//     Term 143 (AT2000-0250)/Term 144 (AT2000-5250)/FB Inputs/Value Channel 06 <-> Data Pointer/RawPositionValues[5]
//     Term 143 (AT2000-0250)/Term 144 (AT2000-5250)/FB Inputs/Value Channel 07 <-> Data Pointer/RawPositionValues[6]
//     Term 143 (AT2000-0250)/Term 144 (AT2000-5250)/FB Inputs/Value Channel 08 <-> Data Pointer/RawPositionValues[7]
//     Term 143 (AT2000-0250)/Term 144 (AT2000-5250)/FB Inputs/Value Channel 09 <-> Data Pointer/RawPositionValues[8]
//     Term 143 (AT2000-0250)/Term 144 (AT2000-5250)/FB Inputs/Value Channel 10 <-> Data Pointer/RawPositionValues[9]
//     Term 143 (AT2000-0250)/Term 144 (AT2000-5250)/FB Inputs/Value Channel 11 <-> Data Pointer/RawPositionValues[10]
//     Term 143 (AT2000-0250)/Term 144 (AT2000-5250)/FB Inputs/Value Channel 12 <-> Data Pointer/RawPositionValues[11]
//     Term 143 (AT2000-0250)/Term 144 (AT2000-5250)/FB Inputs/Value Channel 13 <-> Data Pointer/RawPositionValues[12]
//     Term 143 (AT2000-0250)/Term 144 (AT2000-5250)/FB Inputs/Value Channel 14 <-> Data Pointer/RawPositionValues[13]
//     Term 143 (AT2000-0250)/Term 144 (AT2000-5250)/FB Inputs/Value Channel 15 <-> Data Pointer/RawPositionValues[14]
//     Term 143 (AT2000-0250)/Term 144 (AT2000-5250)/FB Inputs/Value Channel 16 <-> Data Pointer/RawPositionValues[15]
//     Term 143 (AT2000-0250)/Term 144 (AT2000-5250)/FB Inputs/Value Channel 17 <-> Data Pointer/RawPositionValues[16]
//     Term 143 (AT2000-0250)/Term 144 (AT2000-5250)/FB Inputs/Value Channel 18 <-> Data Pointer/RawPositionValues[17]
//     Term 143 (AT2000-0250)/Term 144 (AT2000-5250)/FB Inputs/Value Channel 19 <-> Data Pointer/RawPositionValues[18]
//     Term 143 (AT2000-0250)/Term 144 (AT2000-5250)/FB Inputs/Value Channel 20 <-> Data Pointer/RawPositionValues[19]
//     Term 143 (AT2000-0250)/Term 144 (AT2000-5250)/FB Inputs/Value Channel 21 <-> Data Pointer/RawPositionValues[20]
//     Term 143 (AT2000-0250)/Term 144 (AT2000-5250)/FB Inputs/Value Channel 22 <-> Data Pointer/RawPositionValues[21]
//     Term 143 (AT2000-0250)/Term 144 (AT2000-5250)/FB Inputs/Value Channel 23 <-> Data Pointer/RawPositionValues[22]
//     Term 143 (AT2000-0250)/Term 144 (AT2000-5250)/FB Inputs/Value Channel 24 <-> Data Pointer/RawPositionValues[23]
//     Term 143 (AT2000-0250)/Term 144 (AT2000-5250)/FB Inputs/Value Channel 25 <-> Data Pointer/RawPositionValues[24]
//     Term 143 (AT2000-0250)/Term 144 (AT2000-5250)/FB Inputs/Value Channel 26 <-> Data Pointer/RawPositionValues[25]
//     Term 143 (AT2000-0250)/Term 144 (AT2000-5250)/FB Inputs/Value Channel 27 <-> Data Pointer/RawPositionValues[26]
//     Term 143 (AT2000-0250)/Term 144 (AT2000-5250)/FB Inputs/Value Channel 28 <-> Data Pointer/RawPositionValues[27]
//     Term 143 (AT2000-0250)/Term 144 (AT2000-5250)/FB Inputs/Value Channel 29 <-> Data Pointer/RawPositionValues[28]
//     Term 143 (AT2000-0250)/Term 144 (AT2000-5250)/FB Inputs/Value Channel 30 <-> Data Pointer/RawPositionValues[29]
//     Term 143 (AT2000-0250)/Term 144 (AT2000-5250)/FB Inputs/Value Channel 31 <-> Data Pointer/RawPositionValues[30]
//     Term 143 (AT2000-0250)/Term 144 (AT2000-5250)/FB Inputs/Value Channel 32 <-> Data Pointer/RawPositionValues[31]
//   Device 17 <-> TcCOM Objects/XTS ProcessingUnit 1/Part 1/Module 73
//     Term 145 (AT2000-0250)/CC Inputs/Current actual value Ch.1 <-> Data Pointer/CurrentActualValues[0]
//     Term 145 (AT2000-0250)/CC Inputs/Current actual value Ch.10 <-> Data Pointer/CurrentActualValues[9]
//     Term 145 (AT2000-0250)/CC Inputs/Current actual value Ch.11 <-> Data Pointer/CurrentActualValues[10]
//     Term 145 (AT2000-0250)/CC Inputs/Current actual value Ch.12 <-> Data Pointer/CurrentActualValues[11]
//     Term 145 (AT2000-0250)/CC Inputs/Current actual value Ch.13 <-> Data Pointer/CurrentActualValues[12]
//     Term 145 (AT2000-0250)/CC Inputs/Current actual value Ch.14 <-> Data Pointer/CurrentActualValues[13]
//     Term 145 (AT2000-0250)/CC Inputs/Current actual value Ch.15 <-> Data Pointer/CurrentActualValues[14]
//     Term 145 (AT2000-0250)/CC Inputs/Current actual value Ch.2 <-> Data Pointer/CurrentActualValues[1]
//     Term 145 (AT2000-0250)/CC Inputs/Current actual value Ch.3 <-> Data Pointer/CurrentActualValues[2]
//     Term 145 (AT2000-0250)/CC Inputs/Current actual value Ch.4 <-> Data Pointer/CurrentActualValues[3]
//     Term 145 (AT2000-0250)/CC Inputs/Current actual value Ch.5 <-> Data Pointer/CurrentActualValues[4]
//     Term 145 (AT2000-0250)/CC Inputs/Current actual value Ch.6 <-> Data Pointer/CurrentActualValues[5]
//     Term 145 (AT2000-0250)/CC Inputs/Current actual value Ch.7 <-> Data Pointer/CurrentActualValues[6]
//     Term 145 (AT2000-0250)/CC Inputs/Current actual value Ch.8 <-> Data Pointer/CurrentActualValues[7]
//     Term 145 (AT2000-0250)/CC Inputs/Current actual value Ch.9 <-> Data Pointer/CurrentActualValues[8]
//     Term 145 (AT2000-0250)/CC Inputs/Status <-> Data Pointer/Status
//     Term 145 (AT2000-0250)/CC Outputs/Control <-> Data Pointer/Control
//     Term 145 (AT2000-0250)/CC Outputs/Current setpoint value Ch.1 <-> Data Pointer/CurrentSetpointValues[0]
//     Term 145 (AT2000-0250)/CC Outputs/Current setpoint value Ch.10 <-> Data Pointer/CurrentSetpointValues[9]
//     Term 145 (AT2000-0250)/CC Outputs/Current setpoint value Ch.11 <-> Data Pointer/CurrentSetpointValues[10]
//     Term 145 (AT2000-0250)/CC Outputs/Current setpoint value Ch.12 <-> Data Pointer/CurrentSetpointValues[11]
//     Term 145 (AT2000-0250)/CC Outputs/Current setpoint value Ch.13 <-> Data Pointer/CurrentSetpointValues[12]
//     Term 145 (AT2000-0250)/CC Outputs/Current setpoint value Ch.14 <-> Data Pointer/CurrentSetpointValues[13]
//     Term 145 (AT2000-0250)/CC Outputs/Current setpoint value Ch.15 <-> Data Pointer/CurrentSetpointValues[14]
//     Term 145 (AT2000-0250)/CC Outputs/Current setpoint value Ch.2 <-> Data Pointer/CurrentSetpointValues[1]
//     Term 145 (AT2000-0250)/CC Outputs/Current setpoint value Ch.3 <-> Data Pointer/CurrentSetpointValues[2]
//     Term 145 (AT2000-0250)/CC Outputs/Current setpoint value Ch.4 <-> Data Pointer/CurrentSetpointValues[3]
//     Term 145 (AT2000-0250)/CC Outputs/Current setpoint value Ch.5 <-> Data Pointer/CurrentSetpointValues[4]
//     Term 145 (AT2000-0250)/CC Outputs/Current setpoint value Ch.6 <-> Data Pointer/CurrentSetpointValues[5]
//     Term 145 (AT2000-0250)/CC Outputs/Current setpoint value Ch.7 <-> Data Pointer/CurrentSetpointValues[6]
//     Term 145 (AT2000-0250)/CC Outputs/Current setpoint value Ch.8 <-> Data Pointer/CurrentSetpointValues[7]
//     Term 145 (AT2000-0250)/CC Outputs/Current setpoint value Ch.9 <-> Data Pointer/CurrentSetpointValues[8]
//     Term 145 (AT2000-0250)/Term 146 (AT2000-5250)/FB Inputs/Value Channel 01 <-> Data Pointer/RawPositionValues[0]
//     Term 145 (AT2000-0250)/Term 146 (AT2000-5250)/FB Inputs/Value Channel 02 <-> Data Pointer/RawPositionValues[1]
//     Term 145 (AT2000-0250)/Term 146 (AT2000-5250)/FB Inputs/Value Channel 03 <-> Data Pointer/RawPositionValues[2]
//     Term 145 (AT2000-0250)/Term 146 (AT2000-5250)/FB Inputs/Value Channel 04 <-> Data Pointer/RawPositionValues[3]
//     Term 145 (AT2000-0250)/Term 146 (AT2000-5250)/FB Inputs/Value Channel 05 <-> Data Pointer/RawPositionValues[4]
//     Term 145 (AT2000-0250)/Term 146 (AT2000-5250)/FB Inputs/Value Channel 06 <-> Data Pointer/RawPositionValues[5]
//     Term 145 (AT2000-0250)/Term 146 (AT2000-5250)/FB Inputs/Value Channel 07 <-> Data Pointer/RawPositionValues[6]
//     Term 145 (AT2000-0250)/Term 146 (AT2000-5250)/FB Inputs/Value Channel 08 <-> Data Pointer/RawPositionValues[7]
//     Term 145 (AT2000-0250)/Term 146 (AT2000-5250)/FB Inputs/Value Channel 09 <-> Data Pointer/RawPositionValues[8]
//     Term 145 (AT2000-0250)/Term 146 (AT2000-5250)/FB Inputs/Value Channel 10 <-> Data Pointer/RawPositionValues[9]
//     Term 145 (AT2000-0250)/Term 146 (AT2000-5250)/FB Inputs/Value Channel 11 <-> Data Pointer/RawPositionValues[10]
//     Term 145 (AT2000-0250)/Term 146 (AT2000-5250)/FB Inputs/Value Channel 12 <-> Data Pointer/RawPositionValues[11]
//     Term 145 (AT2000-0250)/Term 146 (AT2000-5250)/FB Inputs/Value Channel 13 <-> Data Pointer/RawPositionValues[12]
//     Term 145 (AT2000-0250)/Term 146 (AT2000-5250)/FB Inputs/Value Channel 14 <-> Data Pointer/RawPositionValues[13]
//     Term 145 (AT2000-0250)/Term 146 (AT2000-5250)/FB Inputs/Value Channel 15 <-> Data Pointer/RawPositionValues[14]
//     Term 145 (AT2000-0250)/Term 146 (AT2000-5250)/FB Inputs/Value Channel 16 <-> Data Pointer/RawPositionValues[15]
//     Term 145 (AT2000-0250)/Term 146 (AT2000-5250)/FB Inputs/Value Channel 17 <-> Data Pointer/RawPositionValues[16]
//     Term 145 (AT2000-0250)/Term 146 (AT2000-5250)/FB Inputs/Value Channel 18 <-> Data Pointer/RawPositionValues[17]
//     Term 145 (AT2000-0250)/Term 146 (AT2000-5250)/FB Inputs/Value Channel 19 <-> Data Pointer/RawPositionValues[18]
//     Term 145 (AT2000-0250)/Term 146 (AT2000-5250)/FB Inputs/Value Channel 20 <-> Data Pointer/RawPositionValues[19]
//     Term 145 (AT2000-0250)/Term 146 (AT2000-5250)/FB Inputs/Value Channel 21 <-> Data Pointer/RawPositionValues[20]
//     Term 145 (AT2000-0250)/Term 146 (AT2000-5250)/FB Inputs/Value Channel 22 <-> Data Pointer/RawPositionValues[21]
//     Term 145 (AT2000-0250)/Term 146 (AT2000-5250)/FB Inputs/Value Channel 23 <-> Data Pointer/RawPositionValues[22]
//     Term 145 (AT2000-0250)/Term 146 (AT2000-5250)/FB Inputs/Value Channel 24 <-> Data Pointer/RawPositionValues[23]
//     Term 145 (AT2000-0250)/Term 146 (AT2000-5250)/FB Inputs/Value Channel 25 <-> Data Pointer/RawPositionValues[24]
//     Term 145 (AT2000-0250)/Term 146 (AT2000-5250)/FB Inputs/Value Channel 26 <-> Data Pointer/RawPositionValues[25]
//     Term 145 (AT2000-0250)/Term 146 (AT2000-5250)/FB Inputs/Value Channel 27 <-> Data Pointer/RawPositionValues[26]
//     Term 145 (AT2000-0250)/Term 146 (AT2000-5250)/FB Inputs/Value Channel 28 <-> Data Pointer/RawPositionValues[27]
//     Term 145 (AT2000-0250)/Term 146 (AT2000-5250)/FB Inputs/Value Channel 29 <-> Data Pointer/RawPositionValues[28]
//     Term 145 (AT2000-0250)/Term 146 (AT2000-5250)/FB Inputs/Value Channel 30 <-> Data Pointer/RawPositionValues[29]
//     Term 145 (AT2000-0250)/Term 146 (AT2000-5250)/FB Inputs/Value Channel 31 <-> Data Pointer/RawPositionValues[30]
//     Term 145 (AT2000-0250)/Term 146 (AT2000-5250)/FB Inputs/Value Channel 32 <-> Data Pointer/RawPositionValues[31]
//   Device 18 <-> TcCOM Objects/XTS ProcessingUnit 1/Part 1/Module 74
//     Term 147 (AT2002-0250)/CC Inputs/Current actual value Ch.1 <-> Data Pointer/CurrentActualValues[0]
//     Term 147 (AT2002-0250)/CC Inputs/Current actual value Ch.10 <-> Data Pointer/CurrentActualValues[9]
//     Term 147 (AT2002-0250)/CC Inputs/Current actual value Ch.11 <-> Data Pointer/CurrentActualValues[10]
//     Term 147 (AT2002-0250)/CC Inputs/Current actual value Ch.12 <-> Data Pointer/CurrentActualValues[11]
//     Term 147 (AT2002-0250)/CC Inputs/Current actual value Ch.13 <-> Data Pointer/CurrentActualValues[12]
//     Term 147 (AT2002-0250)/CC Inputs/Current actual value Ch.14 <-> Data Pointer/CurrentActualValues[13]
//     Term 147 (AT2002-0250)/CC Inputs/Current actual value Ch.15 <-> Data Pointer/CurrentActualValues[14]
//     Term 147 (AT2002-0250)/CC Inputs/Current actual value Ch.2 <-> Data Pointer/CurrentActualValues[1]
//     Term 147 (AT2002-0250)/CC Inputs/Current actual value Ch.3 <-> Data Pointer/CurrentActualValues[2]
//     Term 147 (AT2002-0250)/CC Inputs/Current actual value Ch.4 <-> Data Pointer/CurrentActualValues[3]
//     Term 147 (AT2002-0250)/CC Inputs/Current actual value Ch.5 <-> Data Pointer/CurrentActualValues[4]
//     Term 147 (AT2002-0250)/CC Inputs/Current actual value Ch.6 <-> Data Pointer/CurrentActualValues[5]
//     Term 147 (AT2002-0250)/CC Inputs/Current actual value Ch.7 <-> Data Pointer/CurrentActualValues[6]
//     Term 147 (AT2002-0250)/CC Inputs/Current actual value Ch.8 <-> Data Pointer/CurrentActualValues[7]
//     Term 147 (AT2002-0250)/CC Inputs/Current actual value Ch.9 <-> Data Pointer/CurrentActualValues[8]
//     Term 147 (AT2002-0250)/CC Inputs/Status <-> Data Pointer/Status
//     Term 147 (AT2002-0250)/CC Outputs/Control <-> Data Pointer/Control
//     Term 147 (AT2002-0250)/CC Outputs/Current setpoint value Ch.1 <-> Data Pointer/CurrentSetpointValues[0]
//     Term 147 (AT2002-0250)/CC Outputs/Current setpoint value Ch.10 <-> Data Pointer/CurrentSetpointValues[9]
//     Term 147 (AT2002-0250)/CC Outputs/Current setpoint value Ch.11 <-> Data Pointer/CurrentSetpointValues[10]
//     Term 147 (AT2002-0250)/CC Outputs/Current setpoint value Ch.12 <-> Data Pointer/CurrentSetpointValues[11]
//     Term 147 (AT2002-0250)/CC Outputs/Current setpoint value Ch.13 <-> Data Pointer/CurrentSetpointValues[12]
//     Term 147 (AT2002-0250)/CC Outputs/Current setpoint value Ch.14 <-> Data Pointer/CurrentSetpointValues[13]
//     Term 147 (AT2002-0250)/CC Outputs/Current setpoint value Ch.15 <-> Data Pointer/CurrentSetpointValues[14]
//     Term 147 (AT2002-0250)/CC Outputs/Current setpoint value Ch.2 <-> Data Pointer/CurrentSetpointValues[1]
//     Term 147 (AT2002-0250)/CC Outputs/Current setpoint value Ch.3 <-> Data Pointer/CurrentSetpointValues[2]
//     Term 147 (AT2002-0250)/CC Outputs/Current setpoint value Ch.4 <-> Data Pointer/CurrentSetpointValues[3]
//     Term 147 (AT2002-0250)/CC Outputs/Current setpoint value Ch.5 <-> Data Pointer/CurrentSetpointValues[4]
//     Term 147 (AT2002-0250)/CC Outputs/Current setpoint value Ch.6 <-> Data Pointer/CurrentSetpointValues[5]
//     Term 147 (AT2002-0250)/CC Outputs/Current setpoint value Ch.7 <-> Data Pointer/CurrentSetpointValues[6]
//     Term 147 (AT2002-0250)/CC Outputs/Current setpoint value Ch.8 <-> Data Pointer/CurrentSetpointValues[7]
//     Term 147 (AT2002-0250)/CC Outputs/Current setpoint value Ch.9 <-> Data Pointer/CurrentSetpointValues[8]
//     Term 147 (AT2002-0250)/Term 148 (AT2002-5250)/FB Inputs/Value Channel 01 <-> Data Pointer/RawPositionValues[0]
//     Term 147 (AT2002-0250)/Term 148 (AT2002-5250)/FB Inputs/Value Channel 02 <-> Data Pointer/RawPositionValues[1]
//     Term 147 (AT2002-0250)/Term 148 (AT2002-5250)/FB Inputs/Value Channel 03 <-> Data Pointer/RawPositionValues[2]
//     Term 147 (AT2002-0250)/Term 148 (AT2002-5250)/FB Inputs/Value Channel 04 <-> Data Pointer/RawPositionValues[3]
//     Term 147 (AT2002-0250)/Term 148 (AT2002-5250)/FB Inputs/Value Channel 05 <-> Data Pointer/RawPositionValues[4]
//     Term 147 (AT2002-0250)/Term 148 (AT2002-5250)/FB Inputs/Value Channel 06 <-> Data Pointer/RawPositionValues[5]
//     Term 147 (AT2002-0250)/Term 148 (AT2002-5250)/FB Inputs/Value Channel 07 <-> Data Pointer/RawPositionValues[6]
//     Term 147 (AT2002-0250)/Term 148 (AT2002-5250)/FB Inputs/Value Channel 08 <-> Data Pointer/RawPositionValues[7]
//     Term 147 (AT2002-0250)/Term 148 (AT2002-5250)/FB Inputs/Value Channel 09 <-> Data Pointer/RawPositionValues[8]
//     Term 147 (AT2002-0250)/Term 148 (AT2002-5250)/FB Inputs/Value Channel 10 <-> Data Pointer/RawPositionValues[9]
//     Term 147 (AT2002-0250)/Term 148 (AT2002-5250)/FB Inputs/Value Channel 11 <-> Data Pointer/RawPositionValues[10]
//     Term 147 (AT2002-0250)/Term 148 (AT2002-5250)/FB Inputs/Value Channel 12 <-> Data Pointer/RawPositionValues[11]
//     Term 147 (AT2002-0250)/Term 148 (AT2002-5250)/FB Inputs/Value Channel 13 <-> Data Pointer/RawPositionValues[12]
//     Term 147 (AT2002-0250)/Term 148 (AT2002-5250)/FB Inputs/Value Channel 14 <-> Data Pointer/RawPositionValues[13]
//     Term 147 (AT2002-0250)/Term 148 (AT2002-5250)/FB Inputs/Value Channel 15 <-> Data Pointer/RawPositionValues[14]
//     Term 147 (AT2002-0250)/Term 148 (AT2002-5250)/FB Inputs/Value Channel 16 <-> Data Pointer/RawPositionValues[15]
//     Term 147 (AT2002-0250)/Term 148 (AT2002-5250)/FB Inputs/Value Channel 17 <-> Data Pointer/RawPositionValues[16]
//     Term 147 (AT2002-0250)/Term 148 (AT2002-5250)/FB Inputs/Value Channel 18 <-> Data Pointer/RawPositionValues[17]
//     Term 147 (AT2002-0250)/Term 148 (AT2002-5250)/FB Inputs/Value Channel 19 <-> Data Pointer/RawPositionValues[18]
//     Term 147 (AT2002-0250)/Term 148 (AT2002-5250)/FB Inputs/Value Channel 20 <-> Data Pointer/RawPositionValues[19]
//     Term 147 (AT2002-0250)/Term 148 (AT2002-5250)/FB Inputs/Value Channel 21 <-> Data Pointer/RawPositionValues[20]
//     Term 147 (AT2002-0250)/Term 148 (AT2002-5250)/FB Inputs/Value Channel 22 <-> Data Pointer/RawPositionValues[21]
//     Term 147 (AT2002-0250)/Term 148 (AT2002-5250)/FB Inputs/Value Channel 23 <-> Data Pointer/RawPositionValues[22]
//     Term 147 (AT2002-0250)/Term 148 (AT2002-5250)/FB Inputs/Value Channel 24 <-> Data Pointer/RawPositionValues[23]
//     Term 147 (AT2002-0250)/Term 148 (AT2002-5250)/FB Inputs/Value Channel 25 <-> Data Pointer/RawPositionValues[24]
//     Term 147 (AT2002-0250)/Term 148 (AT2002-5250)/FB Inputs/Value Channel 26 <-> Data Pointer/RawPositionValues[25]
//     Term 147 (AT2002-0250)/Term 148 (AT2002-5250)/FB Inputs/Value Channel 27 <-> Data Pointer/RawPositionValues[26]
//     Term 147 (AT2002-0250)/Term 148 (AT2002-5250)/FB Inputs/Value Channel 28 <-> Data Pointer/RawPositionValues[27]
//     Term 147 (AT2002-0250)/Term 148 (AT2002-5250)/FB Inputs/Value Channel 29 <-> Data Pointer/RawPositionValues[28]
//     Term 147 (AT2002-0250)/Term 148 (AT2002-5250)/FB Inputs/Value Channel 30 <-> Data Pointer/RawPositionValues[29]
//     Term 147 (AT2002-0250)/Term 148 (AT2002-5250)/FB Inputs/Value Channel 31 <-> Data Pointer/RawPositionValues[30]
//     Term 147 (AT2002-0250)/Term 148 (AT2002-5250)/FB Inputs/Value Channel 32 <-> Data Pointer/RawPositionValues[31]
//   Device 18 <-> TcCOM Objects/XTS ProcessingUnit 1/Part 1/Module 75
//     Term 149 (AT2000-0250)/CC Inputs/Current actual value Ch.1 <-> Data Pointer/CurrentActualValues[0]
//     Term 149 (AT2000-0250)/CC Inputs/Current actual value Ch.10 <-> Data Pointer/CurrentActualValues[9]
//     Term 149 (AT2000-0250)/CC Inputs/Current actual value Ch.11 <-> Data Pointer/CurrentActualValues[10]
//     Term 149 (AT2000-0250)/CC Inputs/Current actual value Ch.12 <-> Data Pointer/CurrentActualValues[11]
//     Term 149 (AT2000-0250)/CC Inputs/Current actual value Ch.13 <-> Data Pointer/CurrentActualValues[12]
//     Term 149 (AT2000-0250)/CC Inputs/Current actual value Ch.14 <-> Data Pointer/CurrentActualValues[13]
//     Term 149 (AT2000-0250)/CC Inputs/Current actual value Ch.15 <-> Data Pointer/CurrentActualValues[14]
//     Term 149 (AT2000-0250)/CC Inputs/Current actual value Ch.2 <-> Data Pointer/CurrentActualValues[1]
//     Term 149 (AT2000-0250)/CC Inputs/Current actual value Ch.3 <-> Data Pointer/CurrentActualValues[2]
//     Term 149 (AT2000-0250)/CC Inputs/Current actual value Ch.4 <-> Data Pointer/CurrentActualValues[3]
//     Term 149 (AT2000-0250)/CC Inputs/Current actual value Ch.5 <-> Data Pointer/CurrentActualValues[4]
//     Term 149 (AT2000-0250)/CC Inputs/Current actual value Ch.6 <-> Data Pointer/CurrentActualValues[5]
//     Term 149 (AT2000-0250)/CC Inputs/Current actual value Ch.7 <-> Data Pointer/CurrentActualValues[6]
//     Term 149 (AT2000-0250)/CC Inputs/Current actual value Ch.8 <-> Data Pointer/CurrentActualValues[7]
//     Term 149 (AT2000-0250)/CC Inputs/Current actual value Ch.9 <-> Data Pointer/CurrentActualValues[8]
//     Term 149 (AT2000-0250)/CC Inputs/Status <-> Data Pointer/Status
//     Term 149 (AT2000-0250)/CC Outputs/Control <-> Data Pointer/Control
//     Term 149 (AT2000-0250)/CC Outputs/Current setpoint value Ch.1 <-> Data Pointer/CurrentSetpointValues[0]
//     Term 149 (AT2000-0250)/CC Outputs/Current setpoint value Ch.10 <-> Data Pointer/CurrentSetpointValues[9]
//     Term 149 (AT2000-0250)/CC Outputs/Current setpoint value Ch.11 <-> Data Pointer/CurrentSetpointValues[10]
//     Term 149 (AT2000-0250)/CC Outputs/Current setpoint value Ch.12 <-> Data Pointer/CurrentSetpointValues[11]
//     Term 149 (AT2000-0250)/CC Outputs/Current setpoint value Ch.13 <-> Data Pointer/CurrentSetpointValues[12]
//     Term 149 (AT2000-0250)/CC Outputs/Current setpoint value Ch.14 <-> Data Pointer/CurrentSetpointValues[13]
//     Term 149 (AT2000-0250)/CC Outputs/Current setpoint value Ch.15 <-> Data Pointer/CurrentSetpointValues[14]
//     Term 149 (AT2000-0250)/CC Outputs/Current setpoint value Ch.2 <-> Data Pointer/CurrentSetpointValues[1]
//     Term 149 (AT2000-0250)/CC Outputs/Current setpoint value Ch.3 <-> Data Pointer/CurrentSetpointValues[2]
//     Term 149 (AT2000-0250)/CC Outputs/Current setpoint value Ch.4 <-> Data Pointer/CurrentSetpointValues[3]
//     Term 149 (AT2000-0250)/CC Outputs/Current setpoint value Ch.5 <-> Data Pointer/CurrentSetpointValues[4]
//     Term 149 (AT2000-0250)/CC Outputs/Current setpoint value Ch.6 <-> Data Pointer/CurrentSetpointValues[5]
//     Term 149 (AT2000-0250)/CC Outputs/Current setpoint value Ch.7 <-> Data Pointer/CurrentSetpointValues[6]
//     Term 149 (AT2000-0250)/CC Outputs/Current setpoint value Ch.8 <-> Data Pointer/CurrentSetpointValues[7]
//     Term 149 (AT2000-0250)/CC Outputs/Current setpoint value Ch.9 <-> Data Pointer/CurrentSetpointValues[8]
//     Term 149 (AT2000-0250)/Term 150 (AT2000-5250)/FB Inputs/Value Channel 01 <-> Data Pointer/RawPositionValues[0]
//     Term 149 (AT2000-0250)/Term 150 (AT2000-5250)/FB Inputs/Value Channel 02 <-> Data Pointer/RawPositionValues[1]
//     Term 149 (AT2000-0250)/Term 150 (AT2000-5250)/FB Inputs/Value Channel 03 <-> Data Pointer/RawPositionValues[2]
//     Term 149 (AT2000-0250)/Term 150 (AT2000-5250)/FB Inputs/Value Channel 04 <-> Data Pointer/RawPositionValues[3]
//     Term 149 (AT2000-0250)/Term 150 (AT2000-5250)/FB Inputs/Value Channel 05 <-> Data Pointer/RawPositionValues[4]
//     Term 149 (AT2000-0250)/Term 150 (AT2000-5250)/FB Inputs/Value Channel 06 <-> Data Pointer/RawPositionValues[5]
//     Term 149 (AT2000-0250)/Term 150 (AT2000-5250)/FB Inputs/Value Channel 07 <-> Data Pointer/RawPositionValues[6]
//     Term 149 (AT2000-0250)/Term 150 (AT2000-5250)/FB Inputs/Value Channel 08 <-> Data Pointer/RawPositionValues[7]
//     Term 149 (AT2000-0250)/Term 150 (AT2000-5250)/FB Inputs/Value Channel 09 <-> Data Pointer/RawPositionValues[8]
//     Term 149 (AT2000-0250)/Term 150 (AT2000-5250)/FB Inputs/Value Channel 10 <-> Data Pointer/RawPositionValues[9]
//     Term 149 (AT2000-0250)/Term 150 (AT2000-5250)/FB Inputs/Value Channel 11 <-> Data Pointer/RawPositionValues[10]
//     Term 149 (AT2000-0250)/Term 150 (AT2000-5250)/FB Inputs/Value Channel 12 <-> Data Pointer/RawPositionValues[11]
//     Term 149 (AT2000-0250)/Term 150 (AT2000-5250)/FB Inputs/Value Channel 13 <-> Data Pointer/RawPositionValues[12]
//     Term 149 (AT2000-0250)/Term 150 (AT2000-5250)/FB Inputs/Value Channel 14 <-> Data Pointer/RawPositionValues[13]
//     Term 149 (AT2000-0250)/Term 150 (AT2000-5250)/FB Inputs/Value Channel 15 <-> Data Pointer/RawPositionValues[14]
//     Term 149 (AT2000-0250)/Term 150 (AT2000-5250)/FB Inputs/Value Channel 16 <-> Data Pointer/RawPositionValues[15]
//     Term 149 (AT2000-0250)/Term 150 (AT2000-5250)/FB Inputs/Value Channel 17 <-> Data Pointer/RawPositionValues[16]
//     Term 149 (AT2000-0250)/Term 150 (AT2000-5250)/FB Inputs/Value Channel 18 <-> Data Pointer/RawPositionValues[17]
//     Term 149 (AT2000-0250)/Term 150 (AT2000-5250)/FB Inputs/Value Channel 19 <-> Data Pointer/RawPositionValues[18]
//     Term 149 (AT2000-0250)/Term 150 (AT2000-5250)/FB Inputs/Value Channel 20 <-> Data Pointer/RawPositionValues[19]
//     Term 149 (AT2000-0250)/Term 150 (AT2000-5250)/FB Inputs/Value Channel 21 <-> Data Pointer/RawPositionValues[20]
//     Term 149 (AT2000-0250)/Term 150 (AT2000-5250)/FB Inputs/Value Channel 22 <-> Data Pointer/RawPositionValues[21]
//     Term 149 (AT2000-0250)/Term 150 (AT2000-5250)/FB Inputs/Value Channel 23 <-> Data Pointer/RawPositionValues[22]
//     Term 149 (AT2000-0250)/Term 150 (AT2000-5250)/FB Inputs/Value Channel 24 <-> Data Pointer/RawPositionValues[23]
//     Term 149 (AT2000-0250)/Term 150 (AT2000-5250)/FB Inputs/Value Channel 25 <-> Data Pointer/RawPositionValues[24]
//     Term 149 (AT2000-0250)/Term 150 (AT2000-5250)/FB Inputs/Value Channel 26 <-> Data Pointer/RawPositionValues[25]
//     Term 149 (AT2000-0250)/Term 150 (AT2000-5250)/FB Inputs/Value Channel 27 <-> Data Pointer/RawPositionValues[26]
//     Term 149 (AT2000-0250)/Term 150 (AT2000-5250)/FB Inputs/Value Channel 28 <-> Data Pointer/RawPositionValues[27]
//     Term 149 (AT2000-0250)/Term 150 (AT2000-5250)/FB Inputs/Value Channel 29 <-> Data Pointer/RawPositionValues[28]
//     Term 149 (AT2000-0250)/Term 150 (AT2000-5250)/FB Inputs/Value Channel 30 <-> Data Pointer/RawPositionValues[29]
//     Term 149 (AT2000-0250)/Term 150 (AT2000-5250)/FB Inputs/Value Channel 31 <-> Data Pointer/RawPositionValues[30]
//     Term 149 (AT2000-0250)/Term 150 (AT2000-5250)/FB Inputs/Value Channel 32 <-> Data Pointer/RawPositionValues[31]
//   Device 18 <-> TcCOM Objects/XTS ProcessingUnit 1/Part 1/Module 76
//     Term 151 (AT2000-0250)/CC Inputs/Current actual value Ch.1 <-> Data Pointer/CurrentActualValues[0]
//     Term 151 (AT2000-0250)/CC Inputs/Current actual value Ch.10 <-> Data Pointer/CurrentActualValues[9]
//     Term 151 (AT2000-0250)/CC Inputs/Current actual value Ch.11 <-> Data Pointer/CurrentActualValues[10]
//     Term 151 (AT2000-0250)/CC Inputs/Current actual value Ch.12 <-> Data Pointer/CurrentActualValues[11]
//     Term 151 (AT2000-0250)/CC Inputs/Current actual value Ch.13 <-> Data Pointer/CurrentActualValues[12]
//     Term 151 (AT2000-0250)/CC Inputs/Current actual value Ch.14 <-> Data Pointer/CurrentActualValues[13]
//     Term 151 (AT2000-0250)/CC Inputs/Current actual value Ch.15 <-> Data Pointer/CurrentActualValues[14]
//     Term 151 (AT2000-0250)/CC Inputs/Current actual value Ch.2 <-> Data Pointer/CurrentActualValues[1]
//     Term 151 (AT2000-0250)/CC Inputs/Current actual value Ch.3 <-> Data Pointer/CurrentActualValues[2]
//     Term 151 (AT2000-0250)/CC Inputs/Current actual value Ch.4 <-> Data Pointer/CurrentActualValues[3]
//     Term 151 (AT2000-0250)/CC Inputs/Current actual value Ch.5 <-> Data Pointer/CurrentActualValues[4]
//     Term 151 (AT2000-0250)/CC Inputs/Current actual value Ch.6 <-> Data Pointer/CurrentActualValues[5]
//     Term 151 (AT2000-0250)/CC Inputs/Current actual value Ch.7 <-> Data Pointer/CurrentActualValues[6]
//     Term 151 (AT2000-0250)/CC Inputs/Current actual value Ch.8 <-> Data Pointer/CurrentActualValues[7]
//     Term 151 (AT2000-0250)/CC Inputs/Current actual value Ch.9 <-> Data Pointer/CurrentActualValues[8]
//     Term 151 (AT2000-0250)/CC Inputs/Status <-> Data Pointer/Status
//     Term 151 (AT2000-0250)/CC Outputs/Control <-> Data Pointer/Control
//     Term 151 (AT2000-0250)/CC Outputs/Current setpoint value Ch.1 <-> Data Pointer/CurrentSetpointValues[0]
//     Term 151 (AT2000-0250)/CC Outputs/Current setpoint value Ch.10 <-> Data Pointer/CurrentSetpointValues[9]
//     Term 151 (AT2000-0250)/CC Outputs/Current setpoint value Ch.11 <-> Data Pointer/CurrentSetpointValues[10]
//     Term 151 (AT2000-0250)/CC Outputs/Current setpoint value Ch.12 <-> Data Pointer/CurrentSetpointValues[11]
//     Term 151 (AT2000-0250)/CC Outputs/Current setpoint value Ch.13 <-> Data Pointer/CurrentSetpointValues[12]
//     Term 151 (AT2000-0250)/CC Outputs/Current setpoint value Ch.14 <-> Data Pointer/CurrentSetpointValues[13]
//     Term 151 (AT2000-0250)/CC Outputs/Current setpoint value Ch.15 <-> Data Pointer/CurrentSetpointValues[14]
//     Term 151 (AT2000-0250)/CC Outputs/Current setpoint value Ch.2 <-> Data Pointer/CurrentSetpointValues[1]
//     Term 151 (AT2000-0250)/CC Outputs/Current setpoint value Ch.3 <-> Data Pointer/CurrentSetpointValues[2]
//     Term 151 (AT2000-0250)/CC Outputs/Current setpoint value Ch.4 <-> Data Pointer/CurrentSetpointValues[3]
//     Term 151 (AT2000-0250)/CC Outputs/Current setpoint value Ch.5 <-> Data Pointer/CurrentSetpointValues[4]
//     Term 151 (AT2000-0250)/CC Outputs/Current setpoint value Ch.6 <-> Data Pointer/CurrentSetpointValues[5]
//     Term 151 (AT2000-0250)/CC Outputs/Current setpoint value Ch.7 <-> Data Pointer/CurrentSetpointValues[6]
//     Term 151 (AT2000-0250)/CC Outputs/Current setpoint value Ch.8 <-> Data Pointer/CurrentSetpointValues[7]
//     Term 151 (AT2000-0250)/CC Outputs/Current setpoint value Ch.9 <-> Data Pointer/CurrentSetpointValues[8]
//     Term 151 (AT2000-0250)/Term 152 (AT2000-5250)/FB Inputs/Value Channel 01 <-> Data Pointer/RawPositionValues[0]
//     Term 151 (AT2000-0250)/Term 152 (AT2000-5250)/FB Inputs/Value Channel 02 <-> Data Pointer/RawPositionValues[1]
//     Term 151 (AT2000-0250)/Term 152 (AT2000-5250)/FB Inputs/Value Channel 03 <-> Data Pointer/RawPositionValues[2]
//     Term 151 (AT2000-0250)/Term 152 (AT2000-5250)/FB Inputs/Value Channel 04 <-> Data Pointer/RawPositionValues[3]
//     Term 151 (AT2000-0250)/Term 152 (AT2000-5250)/FB Inputs/Value Channel 05 <-> Data Pointer/RawPositionValues[4]
//     Term 151 (AT2000-0250)/Term 152 (AT2000-5250)/FB Inputs/Value Channel 06 <-> Data Pointer/RawPositionValues[5]
//     Term 151 (AT2000-0250)/Term 152 (AT2000-5250)/FB Inputs/Value Channel 07 <-> Data Pointer/RawPositionValues[6]
//     Term 151 (AT2000-0250)/Term 152 (AT2000-5250)/FB Inputs/Value Channel 08 <-> Data Pointer/RawPositionValues[7]
//     Term 151 (AT2000-0250)/Term 152 (AT2000-5250)/FB Inputs/Value Channel 09 <-> Data Pointer/RawPositionValues[8]
//     Term 151 (AT2000-0250)/Term 152 (AT2000-5250)/FB Inputs/Value Channel 10 <-> Data Pointer/RawPositionValues[9]
//     Term 151 (AT2000-0250)/Term 152 (AT2000-5250)/FB Inputs/Value Channel 11 <-> Data Pointer/RawPositionValues[10]
//     Term 151 (AT2000-0250)/Term 152 (AT2000-5250)/FB Inputs/Value Channel 12 <-> Data Pointer/RawPositionValues[11]
//     Term 151 (AT2000-0250)/Term 152 (AT2000-5250)/FB Inputs/Value Channel 13 <-> Data Pointer/RawPositionValues[12]
//     Term 151 (AT2000-0250)/Term 152 (AT2000-5250)/FB Inputs/Value Channel 14 <-> Data Pointer/RawPositionValues[13]
//     Term 151 (AT2000-0250)/Term 152 (AT2000-5250)/FB Inputs/Value Channel 15 <-> Data Pointer/RawPositionValues[14]
//     Term 151 (AT2000-0250)/Term 152 (AT2000-5250)/FB Inputs/Value Channel 16 <-> Data Pointer/RawPositionValues[15]
//     Term 151 (AT2000-0250)/Term 152 (AT2000-5250)/FB Inputs/Value Channel 17 <-> Data Pointer/RawPositionValues[16]
//     Term 151 (AT2000-0250)/Term 152 (AT2000-5250)/FB Inputs/Value Channel 18 <-> Data Pointer/RawPositionValues[17]
//     Term 151 (AT2000-0250)/Term 152 (AT2000-5250)/FB Inputs/Value Channel 19 <-> Data Pointer/RawPositionValues[18]
//     Term 151 (AT2000-0250)/Term 152 (AT2000-5250)/FB Inputs/Value Channel 20 <-> Data Pointer/RawPositionValues[19]
//     Term 151 (AT2000-0250)/Term 152 (AT2000-5250)/FB Inputs/Value Channel 21 <-> Data Pointer/RawPositionValues[20]
//     Term 151 (AT2000-0250)/Term 152 (AT2000-5250)/FB Inputs/Value Channel 22 <-> Data Pointer/RawPositionValues[21]
//     Term 151 (AT2000-0250)/Term 152 (AT2000-5250)/FB Inputs/Value Channel 23 <-> Data Pointer/RawPositionValues[22]
//     Term 151 (AT2000-0250)/Term 152 (AT2000-5250)/FB Inputs/Value Channel 24 <-> Data Pointer/RawPositionValues[23]
//     Term 151 (AT2000-0250)/Term 152 (AT2000-5250)/FB Inputs/Value Channel 25 <-> Data Pointer/RawPositionValues[24]
//     Term 151 (AT2000-0250)/Term 152 (AT2000-5250)/FB Inputs/Value Channel 26 <-> Data Pointer/RawPositionValues[25]
//     Term 151 (AT2000-0250)/Term 152 (AT2000-5250)/FB Inputs/Value Channel 27 <-> Data Pointer/RawPositionValues[26]
//     Term 151 (AT2000-0250)/Term 152 (AT2000-5250)/FB Inputs/Value Channel 28 <-> Data Pointer/RawPositionValues[27]
//     Term 151 (AT2000-0250)/Term 152 (AT2000-5250)/FB Inputs/Value Channel 29 <-> Data Pointer/RawPositionValues[28]
//     Term 151 (AT2000-0250)/Term 152 (AT2000-5250)/FB Inputs/Value Channel 30 <-> Data Pointer/RawPositionValues[29]
//     Term 151 (AT2000-0250)/Term 152 (AT2000-5250)/FB Inputs/Value Channel 31 <-> Data Pointer/RawPositionValues[30]
//     Term 151 (AT2000-0250)/Term 152 (AT2000-5250)/FB Inputs/Value Channel 32 <-> Data Pointer/RawPositionValues[31]
//   Device 18 <-> TcCOM Objects/XTS ProcessingUnit 1/Part 1/Module 77
//     Term 153 (AT2000-0250)/CC Inputs/Current actual value Ch.1 <-> Data Pointer/CurrentActualValues[0]
//     Term 153 (AT2000-0250)/CC Inputs/Current actual value Ch.10 <-> Data Pointer/CurrentActualValues[9]
//     Term 153 (AT2000-0250)/CC Inputs/Current actual value Ch.11 <-> Data Pointer/CurrentActualValues[10]
//     Term 153 (AT2000-0250)/CC Inputs/Current actual value Ch.12 <-> Data Pointer/CurrentActualValues[11]
//     Term 153 (AT2000-0250)/CC Inputs/Current actual value Ch.13 <-> Data Pointer/CurrentActualValues[12]
//     Term 153 (AT2000-0250)/CC Inputs/Current actual value Ch.14 <-> Data Pointer/CurrentActualValues[13]
//     Term 153 (AT2000-0250)/CC Inputs/Current actual value Ch.15 <-> Data Pointer/CurrentActualValues[14]
//     Term 153 (AT2000-0250)/CC Inputs/Current actual value Ch.2 <-> Data Pointer/CurrentActualValues[1]
//     Term 153 (AT2000-0250)/CC Inputs/Current actual value Ch.3 <-> Data Pointer/CurrentActualValues[2]
//     Term 153 (AT2000-0250)/CC Inputs/Current actual value Ch.4 <-> Data Pointer/CurrentActualValues[3]
//     Term 153 (AT2000-0250)/CC Inputs/Current actual value Ch.5 <-> Data Pointer/CurrentActualValues[4]
//     Term 153 (AT2000-0250)/CC Inputs/Current actual value Ch.6 <-> Data Pointer/CurrentActualValues[5]
//     Term 153 (AT2000-0250)/CC Inputs/Current actual value Ch.7 <-> Data Pointer/CurrentActualValues[6]
//     Term 153 (AT2000-0250)/CC Inputs/Current actual value Ch.8 <-> Data Pointer/CurrentActualValues[7]
//     Term 153 (AT2000-0250)/CC Inputs/Current actual value Ch.9 <-> Data Pointer/CurrentActualValues[8]
//     Term 153 (AT2000-0250)/CC Inputs/Status <-> Data Pointer/Status
//     Term 153 (AT2000-0250)/CC Outputs/Control <-> Data Pointer/Control
//     Term 153 (AT2000-0250)/CC Outputs/Current setpoint value Ch.1 <-> Data Pointer/CurrentSetpointValues[0]
//     Term 153 (AT2000-0250)/CC Outputs/Current setpoint value Ch.10 <-> Data Pointer/CurrentSetpointValues[9]
//     Term 153 (AT2000-0250)/CC Outputs/Current setpoint value Ch.11 <-> Data Pointer/CurrentSetpointValues[10]
//     Term 153 (AT2000-0250)/CC Outputs/Current setpoint value Ch.12 <-> Data Pointer/CurrentSetpointValues[11]
//     Term 153 (AT2000-0250)/CC Outputs/Current setpoint value Ch.13 <-> Data Pointer/CurrentSetpointValues[12]
//     Term 153 (AT2000-0250)/CC Outputs/Current setpoint value Ch.14 <-> Data Pointer/CurrentSetpointValues[13]
//     Term 153 (AT2000-0250)/CC Outputs/Current setpoint value Ch.15 <-> Data Pointer/CurrentSetpointValues[14]
//     Term 153 (AT2000-0250)/CC Outputs/Current setpoint value Ch.2 <-> Data Pointer/CurrentSetpointValues[1]
//     Term 153 (AT2000-0250)/CC Outputs/Current setpoint value Ch.3 <-> Data Pointer/CurrentSetpointValues[2]
//     Term 153 (AT2000-0250)/CC Outputs/Current setpoint value Ch.4 <-> Data Pointer/CurrentSetpointValues[3]
//     Term 153 (AT2000-0250)/CC Outputs/Current setpoint value Ch.5 <-> Data Pointer/CurrentSetpointValues[4]
//     Term 153 (AT2000-0250)/CC Outputs/Current setpoint value Ch.6 <-> Data Pointer/CurrentSetpointValues[5]
//     Term 153 (AT2000-0250)/CC Outputs/Current setpoint value Ch.7 <-> Data Pointer/CurrentSetpointValues[6]
//     Term 153 (AT2000-0250)/CC Outputs/Current setpoint value Ch.8 <-> Data Pointer/CurrentSetpointValues[7]
//     Term 153 (AT2000-0250)/CC Outputs/Current setpoint value Ch.9 <-> Data Pointer/CurrentSetpointValues[8]
//     Term 153 (AT2000-0250)/Term 154 (AT2000-5250)/FB Inputs/Value Channel 01 <-> Data Pointer/RawPositionValues[0]
//     Term 153 (AT2000-0250)/Term 154 (AT2000-5250)/FB Inputs/Value Channel 02 <-> Data Pointer/RawPositionValues[1]
//     Term 153 (AT2000-0250)/Term 154 (AT2000-5250)/FB Inputs/Value Channel 03 <-> Data Pointer/RawPositionValues[2]
//     Term 153 (AT2000-0250)/Term 154 (AT2000-5250)/FB Inputs/Value Channel 04 <-> Data Pointer/RawPositionValues[3]
//     Term 153 (AT2000-0250)/Term 154 (AT2000-5250)/FB Inputs/Value Channel 05 <-> Data Pointer/RawPositionValues[4]
//     Term 153 (AT2000-0250)/Term 154 (AT2000-5250)/FB Inputs/Value Channel 06 <-> Data Pointer/RawPositionValues[5]
//     Term 153 (AT2000-0250)/Term 154 (AT2000-5250)/FB Inputs/Value Channel 07 <-> Data Pointer/RawPositionValues[6]
//     Term 153 (AT2000-0250)/Term 154 (AT2000-5250)/FB Inputs/Value Channel 08 <-> Data Pointer/RawPositionValues[7]
//     Term 153 (AT2000-0250)/Term 154 (AT2000-5250)/FB Inputs/Value Channel 09 <-> Data Pointer/RawPositionValues[8]
//     Term 153 (AT2000-0250)/Term 154 (AT2000-5250)/FB Inputs/Value Channel 10 <-> Data Pointer/RawPositionValues[9]
//     Term 153 (AT2000-0250)/Term 154 (AT2000-5250)/FB Inputs/Value Channel 11 <-> Data Pointer/RawPositionValues[10]
//     Term 153 (AT2000-0250)/Term 154 (AT2000-5250)/FB Inputs/Value Channel 12 <-> Data Pointer/RawPositionValues[11]
//     Term 153 (AT2000-0250)/Term 154 (AT2000-5250)/FB Inputs/Value Channel 13 <-> Data Pointer/RawPositionValues[12]
//     Term 153 (AT2000-0250)/Term 154 (AT2000-5250)/FB Inputs/Value Channel 14 <-> Data Pointer/RawPositionValues[13]
//     Term 153 (AT2000-0250)/Term 154 (AT2000-5250)/FB Inputs/Value Channel 15 <-> Data Pointer/RawPositionValues[14]
//     Term 153 (AT2000-0250)/Term 154 (AT2000-5250)/FB Inputs/Value Channel 16 <-> Data Pointer/RawPositionValues[15]
//     Term 153 (AT2000-0250)/Term 154 (AT2000-5250)/FB Inputs/Value Channel 17 <-> Data Pointer/RawPositionValues[16]
//     Term 153 (AT2000-0250)/Term 154 (AT2000-5250)/FB Inputs/Value Channel 18 <-> Data Pointer/RawPositionValues[17]
//     Term 153 (AT2000-0250)/Term 154 (AT2000-5250)/FB Inputs/Value Channel 19 <-> Data Pointer/RawPositionValues[18]
//     Term 153 (AT2000-0250)/Term 154 (AT2000-5250)/FB Inputs/Value Channel 20 <-> Data Pointer/RawPositionValues[19]
//     Term 153 (AT2000-0250)/Term 154 (AT2000-5250)/FB Inputs/Value Channel 21 <-> Data Pointer/RawPositionValues[20]
//     Term 153 (AT2000-0250)/Term 154 (AT2000-5250)/FB Inputs/Value Channel 22 <-> Data Pointer/RawPositionValues[21]
//     Term 153 (AT2000-0250)/Term 154 (AT2000-5250)/FB Inputs/Value Channel 23 <-> Data Pointer/RawPositionValues[22]
//     Term 153 (AT2000-0250)/Term 154 (AT2000-5250)/FB Inputs/Value Channel 24 <-> Data Pointer/RawPositionValues[23]
//     Term 153 (AT2000-0250)/Term 154 (AT2000-5250)/FB Inputs/Value Channel 25 <-> Data Pointer/RawPositionValues[24]
//     Term 153 (AT2000-0250)/Term 154 (AT2000-5250)/FB Inputs/Value Channel 26 <-> Data Pointer/RawPositionValues[25]
//     Term 153 (AT2000-0250)/Term 154 (AT2000-5250)/FB Inputs/Value Channel 27 <-> Data Pointer/RawPositionValues[26]
//     Term 153 (AT2000-0250)/Term 154 (AT2000-5250)/FB Inputs/Value Channel 28 <-> Data Pointer/RawPositionValues[27]
//     Term 153 (AT2000-0250)/Term 154 (AT2000-5250)/FB Inputs/Value Channel 29 <-> Data Pointer/RawPositionValues[28]
//     Term 153 (AT2000-0250)/Term 154 (AT2000-5250)/FB Inputs/Value Channel 30 <-> Data Pointer/RawPositionValues[29]
//     Term 153 (AT2000-0250)/Term 154 (AT2000-5250)/FB Inputs/Value Channel 31 <-> Data Pointer/RawPositionValues[30]
//     Term 153 (AT2000-0250)/Term 154 (AT2000-5250)/FB Inputs/Value Channel 32 <-> Data Pointer/RawPositionValues[31]
//   Device 18 <-> TcCOM Objects/XTS ProcessingUnit 1/Part 1/Module 78
//     Term 155 (AT2000-0250)/CC Inputs/Current actual value Ch.1 <-> Data Pointer/CurrentActualValues[0]
//     Term 155 (AT2000-0250)/CC Inputs/Current actual value Ch.10 <-> Data Pointer/CurrentActualValues[9]
//     Term 155 (AT2000-0250)/CC Inputs/Current actual value Ch.11 <-> Data Pointer/CurrentActualValues[10]
//     Term 155 (AT2000-0250)/CC Inputs/Current actual value Ch.12 <-> Data Pointer/CurrentActualValues[11]
//     Term 155 (AT2000-0250)/CC Inputs/Current actual value Ch.13 <-> Data Pointer/CurrentActualValues[12]
//     Term 155 (AT2000-0250)/CC Inputs/Current actual value Ch.14 <-> Data Pointer/CurrentActualValues[13]
//     Term 155 (AT2000-0250)/CC Inputs/Current actual value Ch.15 <-> Data Pointer/CurrentActualValues[14]
//     Term 155 (AT2000-0250)/CC Inputs/Current actual value Ch.2 <-> Data Pointer/CurrentActualValues[1]
//     Term 155 (AT2000-0250)/CC Inputs/Current actual value Ch.3 <-> Data Pointer/CurrentActualValues[2]
//     Term 155 (AT2000-0250)/CC Inputs/Current actual value Ch.4 <-> Data Pointer/CurrentActualValues[3]
//     Term 155 (AT2000-0250)/CC Inputs/Current actual value Ch.5 <-> Data Pointer/CurrentActualValues[4]
//     Term 155 (AT2000-0250)/CC Inputs/Current actual value Ch.6 <-> Data Pointer/CurrentActualValues[5]
//     Term 155 (AT2000-0250)/CC Inputs/Current actual value Ch.7 <-> Data Pointer/CurrentActualValues[6]
//     Term 155 (AT2000-0250)/CC Inputs/Current actual value Ch.8 <-> Data Pointer/CurrentActualValues[7]
//     Term 155 (AT2000-0250)/CC Inputs/Current actual value Ch.9 <-> Data Pointer/CurrentActualValues[8]
//     Term 155 (AT2000-0250)/CC Inputs/Status <-> Data Pointer/Status
//     Term 155 (AT2000-0250)/CC Outputs/Control <-> Data Pointer/Control
//     Term 155 (AT2000-0250)/CC Outputs/Current setpoint value Ch.1 <-> Data Pointer/CurrentSetpointValues[0]
//     Term 155 (AT2000-0250)/CC Outputs/Current setpoint value Ch.10 <-> Data Pointer/CurrentSetpointValues[9]
//     Term 155 (AT2000-0250)/CC Outputs/Current setpoint value Ch.11 <-> Data Pointer/CurrentSetpointValues[10]
//     Term 155 (AT2000-0250)/CC Outputs/Current setpoint value Ch.12 <-> Data Pointer/CurrentSetpointValues[11]
//     Term 155 (AT2000-0250)/CC Outputs/Current setpoint value Ch.13 <-> Data Pointer/CurrentSetpointValues[12]
//     Term 155 (AT2000-0250)/CC Outputs/Current setpoint value Ch.14 <-> Data Pointer/CurrentSetpointValues[13]
//     Term 155 (AT2000-0250)/CC Outputs/Current setpoint value Ch.15 <-> Data Pointer/CurrentSetpointValues[14]
//     Term 155 (AT2000-0250)/CC Outputs/Current setpoint value Ch.2 <-> Data Pointer/CurrentSetpointValues[1]
//     Term 155 (AT2000-0250)/CC Outputs/Current setpoint value Ch.3 <-> Data Pointer/CurrentSetpointValues[2]
//     Term 155 (AT2000-0250)/CC Outputs/Current setpoint value Ch.4 <-> Data Pointer/CurrentSetpointValues[3]
//     Term 155 (AT2000-0250)/CC Outputs/Current setpoint value Ch.5 <-> Data Pointer/CurrentSetpointValues[4]
//     Term 155 (AT2000-0250)/CC Outputs/Current setpoint value Ch.6 <-> Data Pointer/CurrentSetpointValues[5]
//     Term 155 (AT2000-0250)/CC Outputs/Current setpoint value Ch.7 <-> Data Pointer/CurrentSetpointValues[6]
//     Term 155 (AT2000-0250)/CC Outputs/Current setpoint value Ch.8 <-> Data Pointer/CurrentSetpointValues[7]
//     Term 155 (AT2000-0250)/CC Outputs/Current setpoint value Ch.9 <-> Data Pointer/CurrentSetpointValues[8]
//     Term 155 (AT2000-0250)/Term 156 (AT2000-5250)/FB Inputs/Value Channel 01 <-> Data Pointer/RawPositionValues[0]
//     Term 155 (AT2000-0250)/Term 156 (AT2000-5250)/FB Inputs/Value Channel 02 <-> Data Pointer/RawPositionValues[1]
//     Term 155 (AT2000-0250)/Term 156 (AT2000-5250)/FB Inputs/Value Channel 03 <-> Data Pointer/RawPositionValues[2]
//     Term 155 (AT2000-0250)/Term 156 (AT2000-5250)/FB Inputs/Value Channel 04 <-> Data Pointer/RawPositionValues[3]
//     Term 155 (AT2000-0250)/Term 156 (AT2000-5250)/FB Inputs/Value Channel 05 <-> Data Pointer/RawPositionValues[4]
//     Term 155 (AT2000-0250)/Term 156 (AT2000-5250)/FB Inputs/Value Channel 06 <-> Data Pointer/RawPositionValues[5]
//     Term 155 (AT2000-0250)/Term 156 (AT2000-5250)/FB Inputs/Value Channel 07 <-> Data Pointer/RawPositionValues[6]
//     Term 155 (AT2000-0250)/Term 156 (AT2000-5250)/FB Inputs/Value Channel 08 <-> Data Pointer/RawPositionValues[7]
//     Term 155 (AT2000-0250)/Term 156 (AT2000-5250)/FB Inputs/Value Channel 09 <-> Data Pointer/RawPositionValues[8]
//     Term 155 (AT2000-0250)/Term 156 (AT2000-5250)/FB Inputs/Value Channel 10 <-> Data Pointer/RawPositionValues[9]
//     Term 155 (AT2000-0250)/Term 156 (AT2000-5250)/FB Inputs/Value Channel 11 <-> Data Pointer/RawPositionValues[10]
//     Term 155 (AT2000-0250)/Term 156 (AT2000-5250)/FB Inputs/Value Channel 12 <-> Data Pointer/RawPositionValues[11]
//     Term 155 (AT2000-0250)/Term 156 (AT2000-5250)/FB Inputs/Value Channel 13 <-> Data Pointer/RawPositionValues[12]
//     Term 155 (AT2000-0250)/Term 156 (AT2000-5250)/FB Inputs/Value Channel 14 <-> Data Pointer/RawPositionValues[13]
//     Term 155 (AT2000-0250)/Term 156 (AT2000-5250)/FB Inputs/Value Channel 15 <-> Data Pointer/RawPositionValues[14]
//     Term 155 (AT2000-0250)/Term 156 (AT2000-5250)/FB Inputs/Value Channel 16 <-> Data Pointer/RawPositionValues[15]
//     Term 155 (AT2000-0250)/Term 156 (AT2000-5250)/FB Inputs/Value Channel 17 <-> Data Pointer/RawPositionValues[16]
//     Term 155 (AT2000-0250)/Term 156 (AT2000-5250)/FB Inputs/Value Channel 18 <-> Data Pointer/RawPositionValues[17]
//     Term 155 (AT2000-0250)/Term 156 (AT2000-5250)/FB Inputs/Value Channel 19 <-> Data Pointer/RawPositionValues[18]
//     Term 155 (AT2000-0250)/Term 156 (AT2000-5250)/FB Inputs/Value Channel 20 <-> Data Pointer/RawPositionValues[19]
//     Term 155 (AT2000-0250)/Term 156 (AT2000-5250)/FB Inputs/Value Channel 21 <-> Data Pointer/RawPositionValues[20]
//     Term 155 (AT2000-0250)/Term 156 (AT2000-5250)/FB Inputs/Value Channel 22 <-> Data Pointer/RawPositionValues[21]
//     Term 155 (AT2000-0250)/Term 156 (AT2000-5250)/FB Inputs/Value Channel 23 <-> Data Pointer/RawPositionValues[22]
//     Term 155 (AT2000-0250)/Term 156 (AT2000-5250)/FB Inputs/Value Channel 24 <-> Data Pointer/RawPositionValues[23]
//     Term 155 (AT2000-0250)/Term 156 (AT2000-5250)/FB Inputs/Value Channel 25 <-> Data Pointer/RawPositionValues[24]
//     Term 155 (AT2000-0250)/Term 156 (AT2000-5250)/FB Inputs/Value Channel 26 <-> Data Pointer/RawPositionValues[25]
//     Term 155 (AT2000-0250)/Term 156 (AT2000-5250)/FB Inputs/Value Channel 27 <-> Data Pointer/RawPositionValues[26]
//     Term 155 (AT2000-0250)/Term 156 (AT2000-5250)/FB Inputs/Value Channel 28 <-> Data Pointer/RawPositionValues[27]
//     Term 155 (AT2000-0250)/Term 156 (AT2000-5250)/FB Inputs/Value Channel 29 <-> Data Pointer/RawPositionValues[28]
//     Term 155 (AT2000-0250)/Term 156 (AT2000-5250)/FB Inputs/Value Channel 30 <-> Data Pointer/RawPositionValues[29]
//     Term 155 (AT2000-0250)/Term 156 (AT2000-5250)/FB Inputs/Value Channel 31 <-> Data Pointer/RawPositionValues[30]
//     Term 155 (AT2000-0250)/Term 156 (AT2000-5250)/FB Inputs/Value Channel 32 <-> Data Pointer/RawPositionValues[31]
//   Device 19 <-> TcCOM Objects/XTS ProcessingUnit 1/Part 1/Module 79
//     Term 157 (AT2002-0250)/CC Inputs/Current actual value Ch.1 <-> Data Pointer/CurrentActualValues[0]
//     Term 157 (AT2002-0250)/CC Inputs/Current actual value Ch.10 <-> Data Pointer/CurrentActualValues[9]
//     Term 157 (AT2002-0250)/CC Inputs/Current actual value Ch.11 <-> Data Pointer/CurrentActualValues[10]
//     Term 157 (AT2002-0250)/CC Inputs/Current actual value Ch.12 <-> Data Pointer/CurrentActualValues[11]
//     Term 157 (AT2002-0250)/CC Inputs/Current actual value Ch.13 <-> Data Pointer/CurrentActualValues[12]
//     Term 157 (AT2002-0250)/CC Inputs/Current actual value Ch.14 <-> Data Pointer/CurrentActualValues[13]
//     Term 157 (AT2002-0250)/CC Inputs/Current actual value Ch.15 <-> Data Pointer/CurrentActualValues[14]
//     Term 157 (AT2002-0250)/CC Inputs/Current actual value Ch.2 <-> Data Pointer/CurrentActualValues[1]
//     Term 157 (AT2002-0250)/CC Inputs/Current actual value Ch.3 <-> Data Pointer/CurrentActualValues[2]
//     Term 157 (AT2002-0250)/CC Inputs/Current actual value Ch.4 <-> Data Pointer/CurrentActualValues[3]
//     Term 157 (AT2002-0250)/CC Inputs/Current actual value Ch.5 <-> Data Pointer/CurrentActualValues[4]
//     Term 157 (AT2002-0250)/CC Inputs/Current actual value Ch.6 <-> Data Pointer/CurrentActualValues[5]
//     Term 157 (AT2002-0250)/CC Inputs/Current actual value Ch.7 <-> Data Pointer/CurrentActualValues[6]
//     Term 157 (AT2002-0250)/CC Inputs/Current actual value Ch.8 <-> Data Pointer/CurrentActualValues[7]
//     Term 157 (AT2002-0250)/CC Inputs/Current actual value Ch.9 <-> Data Pointer/CurrentActualValues[8]
//     Term 157 (AT2002-0250)/CC Inputs/Status <-> Data Pointer/Status
//     Term 157 (AT2002-0250)/CC Outputs/Control <-> Data Pointer/Control
//     Term 157 (AT2002-0250)/CC Outputs/Current setpoint value Ch.1 <-> Data Pointer/CurrentSetpointValues[0]
//     Term 157 (AT2002-0250)/CC Outputs/Current setpoint value Ch.10 <-> Data Pointer/CurrentSetpointValues[9]
//     Term 157 (AT2002-0250)/CC Outputs/Current setpoint value Ch.11 <-> Data Pointer/CurrentSetpointValues[10]
//     Term 157 (AT2002-0250)/CC Outputs/Current setpoint value Ch.12 <-> Data Pointer/CurrentSetpointValues[11]
//     Term 157 (AT2002-0250)/CC Outputs/Current setpoint value Ch.13 <-> Data Pointer/CurrentSetpointValues[12]
//     Term 157 (AT2002-0250)/CC Outputs/Current setpoint value Ch.14 <-> Data Pointer/CurrentSetpointValues[13]
//     Term 157 (AT2002-0250)/CC Outputs/Current setpoint value Ch.15 <-> Data Pointer/CurrentSetpointValues[14]
//     Term 157 (AT2002-0250)/CC Outputs/Current setpoint value Ch.2 <-> Data Pointer/CurrentSetpointValues[1]
//     Term 157 (AT2002-0250)/CC Outputs/Current setpoint value Ch.3 <-> Data Pointer/CurrentSetpointValues[2]
//     Term 157 (AT2002-0250)/CC Outputs/Current setpoint value Ch.4 <-> Data Pointer/CurrentSetpointValues[3]
//     Term 157 (AT2002-0250)/CC Outputs/Current setpoint value Ch.5 <-> Data Pointer/CurrentSetpointValues[4]
//     Term 157 (AT2002-0250)/CC Outputs/Current setpoint value Ch.6 <-> Data Pointer/CurrentSetpointValues[5]
//     Term 157 (AT2002-0250)/CC Outputs/Current setpoint value Ch.7 <-> Data Pointer/CurrentSetpointValues[6]
//     Term 157 (AT2002-0250)/CC Outputs/Current setpoint value Ch.8 <-> Data Pointer/CurrentSetpointValues[7]
//     Term 157 (AT2002-0250)/CC Outputs/Current setpoint value Ch.9 <-> Data Pointer/CurrentSetpointValues[8]
//     Term 157 (AT2002-0250)/Term 158 (AT2002-5250)/FB Inputs/Value Channel 01 <-> Data Pointer/RawPositionValues[0]
//     Term 157 (AT2002-0250)/Term 158 (AT2002-5250)/FB Inputs/Value Channel 02 <-> Data Pointer/RawPositionValues[1]
//     Term 157 (AT2002-0250)/Term 158 (AT2002-5250)/FB Inputs/Value Channel 03 <-> Data Pointer/RawPositionValues[2]
//     Term 157 (AT2002-0250)/Term 158 (AT2002-5250)/FB Inputs/Value Channel 04 <-> Data Pointer/RawPositionValues[3]
//     Term 157 (AT2002-0250)/Term 158 (AT2002-5250)/FB Inputs/Value Channel 05 <-> Data Pointer/RawPositionValues[4]
//     Term 157 (AT2002-0250)/Term 158 (AT2002-5250)/FB Inputs/Value Channel 06 <-> Data Pointer/RawPositionValues[5]
//     Term 157 (AT2002-0250)/Term 158 (AT2002-5250)/FB Inputs/Value Channel 07 <-> Data Pointer/RawPositionValues[6]
//     Term 157 (AT2002-0250)/Term 158 (AT2002-5250)/FB Inputs/Value Channel 08 <-> Data Pointer/RawPositionValues[7]
//     Term 157 (AT2002-0250)/Term 158 (AT2002-5250)/FB Inputs/Value Channel 09 <-> Data Pointer/RawPositionValues[8]
//     Term 157 (AT2002-0250)/Term 158 (AT2002-5250)/FB Inputs/Value Channel 10 <-> Data Pointer/RawPositionValues[9]
//     Term 157 (AT2002-0250)/Term 158 (AT2002-5250)/FB Inputs/Value Channel 11 <-> Data Pointer/RawPositionValues[10]
//     Term 157 (AT2002-0250)/Term 158 (AT2002-5250)/FB Inputs/Value Channel 12 <-> Data Pointer/RawPositionValues[11]
//     Term 157 (AT2002-0250)/Term 158 (AT2002-5250)/FB Inputs/Value Channel 13 <-> Data Pointer/RawPositionValues[12]
//     Term 157 (AT2002-0250)/Term 158 (AT2002-5250)/FB Inputs/Value Channel 14 <-> Data Pointer/RawPositionValues[13]
//     Term 157 (AT2002-0250)/Term 158 (AT2002-5250)/FB Inputs/Value Channel 15 <-> Data Pointer/RawPositionValues[14]
//     Term 157 (AT2002-0250)/Term 158 (AT2002-5250)/FB Inputs/Value Channel 16 <-> Data Pointer/RawPositionValues[15]
//     Term 157 (AT2002-0250)/Term 158 (AT2002-5250)/FB Inputs/Value Channel 17 <-> Data Pointer/RawPositionValues[16]
//     Term 157 (AT2002-0250)/Term 158 (AT2002-5250)/FB Inputs/Value Channel 18 <-> Data Pointer/RawPositionValues[17]
//     Term 157 (AT2002-0250)/Term 158 (AT2002-5250)/FB Inputs/Value Channel 19 <-> Data Pointer/RawPositionValues[18]
//     Term 157 (AT2002-0250)/Term 158 (AT2002-5250)/FB Inputs/Value Channel 20 <-> Data Pointer/RawPositionValues[19]
//     Term 157 (AT2002-0250)/Term 158 (AT2002-5250)/FB Inputs/Value Channel 21 <-> Data Pointer/RawPositionValues[20]
//     Term 157 (AT2002-0250)/Term 158 (AT2002-5250)/FB Inputs/Value Channel 22 <-> Data Pointer/RawPositionValues[21]
//     Term 157 (AT2002-0250)/Term 158 (AT2002-5250)/FB Inputs/Value Channel 23 <-> Data Pointer/RawPositionValues[22]
//     Term 157 (AT2002-0250)/Term 158 (AT2002-5250)/FB Inputs/Value Channel 24 <-> Data Pointer/RawPositionValues[23]
//     Term 157 (AT2002-0250)/Term 158 (AT2002-5250)/FB Inputs/Value Channel 25 <-> Data Pointer/RawPositionValues[24]
//     Term 157 (AT2002-0250)/Term 158 (AT2002-5250)/FB Inputs/Value Channel 26 <-> Data Pointer/RawPositionValues[25]
//     Term 157 (AT2002-0250)/Term 158 (AT2002-5250)/FB Inputs/Value Channel 27 <-> Data Pointer/RawPositionValues[26]
//     Term 157 (AT2002-0250)/Term 158 (AT2002-5250)/FB Inputs/Value Channel 28 <-> Data Pointer/RawPositionValues[27]
//     Term 157 (AT2002-0250)/Term 158 (AT2002-5250)/FB Inputs/Value Channel 29 <-> Data Pointer/RawPositionValues[28]
//     Term 157 (AT2002-0250)/Term 158 (AT2002-5250)/FB Inputs/Value Channel 30 <-> Data Pointer/RawPositionValues[29]
//     Term 157 (AT2002-0250)/Term 158 (AT2002-5250)/FB Inputs/Value Channel 31 <-> Data Pointer/RawPositionValues[30]
//     Term 157 (AT2002-0250)/Term 158 (AT2002-5250)/FB Inputs/Value Channel 32 <-> Data Pointer/RawPositionValues[31]
//   Device 19 <-> TcCOM Objects/XTS ProcessingUnit 1/Part 1/Module 80
//     Term 159 (AT2000-0250)/CC Inputs/Current actual value Ch.1 <-> Data Pointer/CurrentActualValues[0]
//     Term 159 (AT2000-0250)/CC Inputs/Current actual value Ch.10 <-> Data Pointer/CurrentActualValues[9]
//     Term 159 (AT2000-0250)/CC Inputs/Current actual value Ch.11 <-> Data Pointer/CurrentActualValues[10]
//     Term 159 (AT2000-0250)/CC Inputs/Current actual value Ch.12 <-> Data Pointer/CurrentActualValues[11]
//     Term 159 (AT2000-0250)/CC Inputs/Current actual value Ch.13 <-> Data Pointer/CurrentActualValues[12]
//     Term 159 (AT2000-0250)/CC Inputs/Current actual value Ch.14 <-> Data Pointer/CurrentActualValues[13]
//     Term 159 (AT2000-0250)/CC Inputs/Current actual value Ch.15 <-> Data Pointer/CurrentActualValues[14]
//     Term 159 (AT2000-0250)/CC Inputs/Current actual value Ch.2 <-> Data Pointer/CurrentActualValues[1]
//     Term 159 (AT2000-0250)/CC Inputs/Current actual value Ch.3 <-> Data Pointer/CurrentActualValues[2]
//     Term 159 (AT2000-0250)/CC Inputs/Current actual value Ch.4 <-> Data Pointer/CurrentActualValues[3]
//     Term 159 (AT2000-0250)/CC Inputs/Current actual value Ch.5 <-> Data Pointer/CurrentActualValues[4]
//     Term 159 (AT2000-0250)/CC Inputs/Current actual value Ch.6 <-> Data Pointer/CurrentActualValues[5]
//     Term 159 (AT2000-0250)/CC Inputs/Current actual value Ch.7 <-> Data Pointer/CurrentActualValues[6]
//     Term 159 (AT2000-0250)/CC Inputs/Current actual value Ch.8 <-> Data Pointer/CurrentActualValues[7]
//     Term 159 (AT2000-0250)/CC Inputs/Current actual value Ch.9 <-> Data Pointer/CurrentActualValues[8]
//     Term 159 (AT2000-0250)/CC Inputs/Status <-> Data Pointer/Status
//     Term 159 (AT2000-0250)/CC Outputs/Control <-> Data Pointer/Control
//     Term 159 (AT2000-0250)/CC Outputs/Current setpoint value Ch.1 <-> Data Pointer/CurrentSetpointValues[0]
//     Term 159 (AT2000-0250)/CC Outputs/Current setpoint value Ch.10 <-> Data Pointer/CurrentSetpointValues[9]
//     Term 159 (AT2000-0250)/CC Outputs/Current setpoint value Ch.11 <-> Data Pointer/CurrentSetpointValues[10]
//     Term 159 (AT2000-0250)/CC Outputs/Current setpoint value Ch.12 <-> Data Pointer/CurrentSetpointValues[11]
//     Term 159 (AT2000-0250)/CC Outputs/Current setpoint value Ch.13 <-> Data Pointer/CurrentSetpointValues[12]
//     Term 159 (AT2000-0250)/CC Outputs/Current setpoint value Ch.14 <-> Data Pointer/CurrentSetpointValues[13]
//     Term 159 (AT2000-0250)/CC Outputs/Current setpoint value Ch.15 <-> Data Pointer/CurrentSetpointValues[14]
//     Term 159 (AT2000-0250)/CC Outputs/Current setpoint value Ch.2 <-> Data Pointer/CurrentSetpointValues[1]
//     Term 159 (AT2000-0250)/CC Outputs/Current setpoint value Ch.3 <-> Data Pointer/CurrentSetpointValues[2]
//     Term 159 (AT2000-0250)/CC Outputs/Current setpoint value Ch.4 <-> Data Pointer/CurrentSetpointValues[3]
//     Term 159 (AT2000-0250)/CC Outputs/Current setpoint value Ch.5 <-> Data Pointer/CurrentSetpointValues[4]
//     Term 159 (AT2000-0250)/CC Outputs/Current setpoint value Ch.6 <-> Data Pointer/CurrentSetpointValues[5]
//     Term 159 (AT2000-0250)/CC Outputs/Current setpoint value Ch.7 <-> Data Pointer/CurrentSetpointValues[6]
//     Term 159 (AT2000-0250)/CC Outputs/Current setpoint value Ch.8 <-> Data Pointer/CurrentSetpointValues[7]
//     Term 159 (AT2000-0250)/CC Outputs/Current setpoint value Ch.9 <-> Data Pointer/CurrentSetpointValues[8]
//     Term 159 (AT2000-0250)/Term 160 (AT2000-5250)/FB Inputs/Value Channel 01 <-> Data Pointer/RawPositionValues[0]
//     Term 159 (AT2000-0250)/Term 160 (AT2000-5250)/FB Inputs/Value Channel 02 <-> Data Pointer/RawPositionValues[1]
//     Term 159 (AT2000-0250)/Term 160 (AT2000-5250)/FB Inputs/Value Channel 03 <-> Data Pointer/RawPositionValues[2]
//     Term 159 (AT2000-0250)/Term 160 (AT2000-5250)/FB Inputs/Value Channel 04 <-> Data Pointer/RawPositionValues[3]
//     Term 159 (AT2000-0250)/Term 160 (AT2000-5250)/FB Inputs/Value Channel 05 <-> Data Pointer/RawPositionValues[4]
//     Term 159 (AT2000-0250)/Term 160 (AT2000-5250)/FB Inputs/Value Channel 06 <-> Data Pointer/RawPositionValues[5]
//     Term 159 (AT2000-0250)/Term 160 (AT2000-5250)/FB Inputs/Value Channel 07 <-> Data Pointer/RawPositionValues[6]
//     Term 159 (AT2000-0250)/Term 160 (AT2000-5250)/FB Inputs/Value Channel 08 <-> Data Pointer/RawPositionValues[7]
//     Term 159 (AT2000-0250)/Term 160 (AT2000-5250)/FB Inputs/Value Channel 09 <-> Data Pointer/RawPositionValues[8]
//     Term 159 (AT2000-0250)/Term 160 (AT2000-5250)/FB Inputs/Value Channel 10 <-> Data Pointer/RawPositionValues[9]
//     Term 159 (AT2000-0250)/Term 160 (AT2000-5250)/FB Inputs/Value Channel 11 <-> Data Pointer/RawPositionValues[10]
//     Term 159 (AT2000-0250)/Term 160 (AT2000-5250)/FB Inputs/Value Channel 12 <-> Data Pointer/RawPositionValues[11]
//     Term 159 (AT2000-0250)/Term 160 (AT2000-5250)/FB Inputs/Value Channel 13 <-> Data Pointer/RawPositionValues[12]
//     Term 159 (AT2000-0250)/Term 160 (AT2000-5250)/FB Inputs/Value Channel 14 <-> Data Pointer/RawPositionValues[13]
//     Term 159 (AT2000-0250)/Term 160 (AT2000-5250)/FB Inputs/Value Channel 15 <-> Data Pointer/RawPositionValues[14]
//     Term 159 (AT2000-0250)/Term 160 (AT2000-5250)/FB Inputs/Value Channel 16 <-> Data Pointer/RawPositionValues[15]
//     Term 159 (AT2000-0250)/Term 160 (AT2000-5250)/FB Inputs/Value Channel 17 <-> Data Pointer/RawPositionValues[16]
//     Term 159 (AT2000-0250)/Term 160 (AT2000-5250)/FB Inputs/Value Channel 18 <-> Data Pointer/RawPositionValues[17]
//     Term 159 (AT2000-0250)/Term 160 (AT2000-5250)/FB Inputs/Value Channel 19 <-> Data Pointer/RawPositionValues[18]
//     Term 159 (AT2000-0250)/Term 160 (AT2000-5250)/FB Inputs/Value Channel 20 <-> Data Pointer/RawPositionValues[19]
//     Term 159 (AT2000-0250)/Term 160 (AT2000-5250)/FB Inputs/Value Channel 21 <-> Data Pointer/RawPositionValues[20]
//     Term 159 (AT2000-0250)/Term 160 (AT2000-5250)/FB Inputs/Value Channel 22 <-> Data Pointer/RawPositionValues[21]
//     Term 159 (AT2000-0250)/Term 160 (AT2000-5250)/FB Inputs/Value Channel 23 <-> Data Pointer/RawPositionValues[22]
//     Term 159 (AT2000-0250)/Term 160 (AT2000-5250)/FB Inputs/Value Channel 24 <-> Data Pointer/RawPositionValues[23]
//     Term 159 (AT2000-0250)/Term 160 (AT2000-5250)/FB Inputs/Value Channel 25 <-> Data Pointer/RawPositionValues[24]
//     Term 159 (AT2000-0250)/Term 160 (AT2000-5250)/FB Inputs/Value Channel 26 <-> Data Pointer/RawPositionValues[25]
//     Term 159 (AT2000-0250)/Term 160 (AT2000-5250)/FB Inputs/Value Channel 27 <-> Data Pointer/RawPositionValues[26]
//     Term 159 (AT2000-0250)/Term 160 (AT2000-5250)/FB Inputs/Value Channel 28 <-> Data Pointer/RawPositionValues[27]
//     Term 159 (AT2000-0250)/Term 160 (AT2000-5250)/FB Inputs/Value Channel 29 <-> Data Pointer/RawPositionValues[28]
//     Term 159 (AT2000-0250)/Term 160 (AT2000-5250)/FB Inputs/Value Channel 30 <-> Data Pointer/RawPositionValues[29]
//     Term 159 (AT2000-0250)/Term 160 (AT2000-5250)/FB Inputs/Value Channel 31 <-> Data Pointer/RawPositionValues[30]
//     Term 159 (AT2000-0250)/Term 160 (AT2000-5250)/FB Inputs/Value Channel 32 <-> Data Pointer/RawPositionValues[31]
//   Device 19 <-> TcCOM Objects/XTS ProcessingUnit 1/Part 1/Module 81
//     Term 161 (AT2000-0250)/CC Inputs/Current actual value Ch.1 <-> Data Pointer/CurrentActualValues[0]
//     Term 161 (AT2000-0250)/CC Inputs/Current actual value Ch.10 <-> Data Pointer/CurrentActualValues[9]
//     Term 161 (AT2000-0250)/CC Inputs/Current actual value Ch.11 <-> Data Pointer/CurrentActualValues[10]
//     Term 161 (AT2000-0250)/CC Inputs/Current actual value Ch.12 <-> Data Pointer/CurrentActualValues[11]
//     Term 161 (AT2000-0250)/CC Inputs/Current actual value Ch.13 <-> Data Pointer/CurrentActualValues[12]
//     Term 161 (AT2000-0250)/CC Inputs/Current actual value Ch.14 <-> Data Pointer/CurrentActualValues[13]
//     Term 161 (AT2000-0250)/CC Inputs/Current actual value Ch.15 <-> Data Pointer/CurrentActualValues[14]
//     Term 161 (AT2000-0250)/CC Inputs/Current actual value Ch.2 <-> Data Pointer/CurrentActualValues[1]
//     Term 161 (AT2000-0250)/CC Inputs/Current actual value Ch.3 <-> Data Pointer/CurrentActualValues[2]
//     Term 161 (AT2000-0250)/CC Inputs/Current actual value Ch.4 <-> Data Pointer/CurrentActualValues[3]
//     Term 161 (AT2000-0250)/CC Inputs/Current actual value Ch.5 <-> Data Pointer/CurrentActualValues[4]
//     Term 161 (AT2000-0250)/CC Inputs/Current actual value Ch.6 <-> Data Pointer/CurrentActualValues[5]
//     Term 161 (AT2000-0250)/CC Inputs/Current actual value Ch.7 <-> Data Pointer/CurrentActualValues[6]
//     Term 161 (AT2000-0250)/CC Inputs/Current actual value Ch.8 <-> Data Pointer/CurrentActualValues[7]
//     Term 161 (AT2000-0250)/CC Inputs/Current actual value Ch.9 <-> Data Pointer/CurrentActualValues[8]
//     Term 161 (AT2000-0250)/CC Inputs/Status <-> Data Pointer/Status
//     Term 161 (AT2000-0250)/CC Outputs/Control <-> Data Pointer/Control
//     Term 161 (AT2000-0250)/CC Outputs/Current setpoint value Ch.1 <-> Data Pointer/CurrentSetpointValues[0]
//     Term 161 (AT2000-0250)/CC Outputs/Current setpoint value Ch.10 <-> Data Pointer/CurrentSetpointValues[9]
//     Term 161 (AT2000-0250)/CC Outputs/Current setpoint value Ch.11 <-> Data Pointer/CurrentSetpointValues[10]
//     Term 161 (AT2000-0250)/CC Outputs/Current setpoint value Ch.12 <-> Data Pointer/CurrentSetpointValues[11]
//     Term 161 (AT2000-0250)/CC Outputs/Current setpoint value Ch.13 <-> Data Pointer/CurrentSetpointValues[12]
//     Term 161 (AT2000-0250)/CC Outputs/Current setpoint value Ch.14 <-> Data Pointer/CurrentSetpointValues[13]
//     Term 161 (AT2000-0250)/CC Outputs/Current setpoint value Ch.15 <-> Data Pointer/CurrentSetpointValues[14]
//     Term 161 (AT2000-0250)/CC Outputs/Current setpoint value Ch.2 <-> Data Pointer/CurrentSetpointValues[1]
//     Term 161 (AT2000-0250)/CC Outputs/Current setpoint value Ch.3 <-> Data Pointer/CurrentSetpointValues[2]
//     Term 161 (AT2000-0250)/CC Outputs/Current setpoint value Ch.4 <-> Data Pointer/CurrentSetpointValues[3]
//     Term 161 (AT2000-0250)/CC Outputs/Current setpoint value Ch.5 <-> Data Pointer/CurrentSetpointValues[4]
//     Term 161 (AT2000-0250)/CC Outputs/Current setpoint value Ch.6 <-> Data Pointer/CurrentSetpointValues[5]
//     Term 161 (AT2000-0250)/CC Outputs/Current setpoint value Ch.7 <-> Data Pointer/CurrentSetpointValues[6]
//     Term 161 (AT2000-0250)/CC Outputs/Current setpoint value Ch.8 <-> Data Pointer/CurrentSetpointValues[7]
//     Term 161 (AT2000-0250)/CC Outputs/Current setpoint value Ch.9 <-> Data Pointer/CurrentSetpointValues[8]
//     Term 161 (AT2000-0250)/Term 162 (AT2000-5250)/FB Inputs/Value Channel 01 <-> Data Pointer/RawPositionValues[0]
//     Term 161 (AT2000-0250)/Term 162 (AT2000-5250)/FB Inputs/Value Channel 02 <-> Data Pointer/RawPositionValues[1]
//     Term 161 (AT2000-0250)/Term 162 (AT2000-5250)/FB Inputs/Value Channel 03 <-> Data Pointer/RawPositionValues[2]
//     Term 161 (AT2000-0250)/Term 162 (AT2000-5250)/FB Inputs/Value Channel 04 <-> Data Pointer/RawPositionValues[3]
//     Term 161 (AT2000-0250)/Term 162 (AT2000-5250)/FB Inputs/Value Channel 05 <-> Data Pointer/RawPositionValues[4]
//     Term 161 (AT2000-0250)/Term 162 (AT2000-5250)/FB Inputs/Value Channel 06 <-> Data Pointer/RawPositionValues[5]
//     Term 161 (AT2000-0250)/Term 162 (AT2000-5250)/FB Inputs/Value Channel 07 <-> Data Pointer/RawPositionValues[6]
//     Term 161 (AT2000-0250)/Term 162 (AT2000-5250)/FB Inputs/Value Channel 08 <-> Data Pointer/RawPositionValues[7]
//     Term 161 (AT2000-0250)/Term 162 (AT2000-5250)/FB Inputs/Value Channel 09 <-> Data Pointer/RawPositionValues[8]
//     Term 161 (AT2000-0250)/Term 162 (AT2000-5250)/FB Inputs/Value Channel 10 <-> Data Pointer/RawPositionValues[9]
//     Term 161 (AT2000-0250)/Term 162 (AT2000-5250)/FB Inputs/Value Channel 11 <-> Data Pointer/RawPositionValues[10]
//     Term 161 (AT2000-0250)/Term 162 (AT2000-5250)/FB Inputs/Value Channel 12 <-> Data Pointer/RawPositionValues[11]
//     Term 161 (AT2000-0250)/Term 162 (AT2000-5250)/FB Inputs/Value Channel 13 <-> Data Pointer/RawPositionValues[12]
//     Term 161 (AT2000-0250)/Term 162 (AT2000-5250)/FB Inputs/Value Channel 14 <-> Data Pointer/RawPositionValues[13]
//     Term 161 (AT2000-0250)/Term 162 (AT2000-5250)/FB Inputs/Value Channel 15 <-> Data Pointer/RawPositionValues[14]
//     Term 161 (AT2000-0250)/Term 162 (AT2000-5250)/FB Inputs/Value Channel 16 <-> Data Pointer/RawPositionValues[15]
//     Term 161 (AT2000-0250)/Term 162 (AT2000-5250)/FB Inputs/Value Channel 17 <-> Data Pointer/RawPositionValues[16]
//     Term 161 (AT2000-0250)/Term 162 (AT2000-5250)/FB Inputs/Value Channel 18 <-> Data Pointer/RawPositionValues[17]
//     Term 161 (AT2000-0250)/Term 162 (AT2000-5250)/FB Inputs/Value Channel 19 <-> Data Pointer/RawPositionValues[18]
//     Term 161 (AT2000-0250)/Term 162 (AT2000-5250)/FB Inputs/Value Channel 20 <-> Data Pointer/RawPositionValues[19]
//     Term 161 (AT2000-0250)/Term 162 (AT2000-5250)/FB Inputs/Value Channel 21 <-> Data Pointer/RawPositionValues[20]
//     Term 161 (AT2000-0250)/Term 162 (AT2000-5250)/FB Inputs/Value Channel 22 <-> Data Pointer/RawPositionValues[21]
//     Term 161 (AT2000-0250)/Term 162 (AT2000-5250)/FB Inputs/Value Channel 23 <-> Data Pointer/RawPositionValues[22]
//     Term 161 (AT2000-0250)/Term 162 (AT2000-5250)/FB Inputs/Value Channel 24 <-> Data Pointer/RawPositionValues[23]
//     Term 161 (AT2000-0250)/Term 162 (AT2000-5250)/FB Inputs/Value Channel 25 <-> Data Pointer/RawPositionValues[24]
//     Term 161 (AT2000-0250)/Term 162 (AT2000-5250)/FB Inputs/Value Channel 26 <-> Data Pointer/RawPositionValues[25]
//     Term 161 (AT2000-0250)/Term 162 (AT2000-5250)/FB Inputs/Value Channel 27 <-> Data Pointer/RawPositionValues[26]
//     Term 161 (AT2000-0250)/Term 162 (AT2000-5250)/FB Inputs/Value Channel 28 <-> Data Pointer/RawPositionValues[27]
//     Term 161 (AT2000-0250)/Term 162 (AT2000-5250)/FB Inputs/Value Channel 29 <-> Data Pointer/RawPositionValues[28]
//     Term 161 (AT2000-0250)/Term 162 (AT2000-5250)/FB Inputs/Value Channel 30 <-> Data Pointer/RawPositionValues[29]
//     Term 161 (AT2000-0250)/Term 162 (AT2000-5250)/FB Inputs/Value Channel 31 <-> Data Pointer/RawPositionValues[30]
//     Term 161 (AT2000-0250)/Term 162 (AT2000-5250)/FB Inputs/Value Channel 32 <-> Data Pointer/RawPositionValues[31]
//   Device 19 <-> TcCOM Objects/XTS ProcessingUnit 1/Part 1/Module 82
//     Term 163 (AT2000-0250)/CC Inputs/Current actual value Ch.1 <-> Data Pointer/CurrentActualValues[0]
//     Term 163 (AT2000-0250)/CC Inputs/Current actual value Ch.10 <-> Data Pointer/CurrentActualValues[9]
//     Term 163 (AT2000-0250)/CC Inputs/Current actual value Ch.11 <-> Data Pointer/CurrentActualValues[10]
//     Term 163 (AT2000-0250)/CC Inputs/Current actual value Ch.12 <-> Data Pointer/CurrentActualValues[11]
//     Term 163 (AT2000-0250)/CC Inputs/Current actual value Ch.13 <-> Data Pointer/CurrentActualValues[12]
//     Term 163 (AT2000-0250)/CC Inputs/Current actual value Ch.14 <-> Data Pointer/CurrentActualValues[13]
//     Term 163 (AT2000-0250)/CC Inputs/Current actual value Ch.15 <-> Data Pointer/CurrentActualValues[14]
//     Term 163 (AT2000-0250)/CC Inputs/Current actual value Ch.2 <-> Data Pointer/CurrentActualValues[1]
//     Term 163 (AT2000-0250)/CC Inputs/Current actual value Ch.3 <-> Data Pointer/CurrentActualValues[2]
//     Term 163 (AT2000-0250)/CC Inputs/Current actual value Ch.4 <-> Data Pointer/CurrentActualValues[3]
//     Term 163 (AT2000-0250)/CC Inputs/Current actual value Ch.5 <-> Data Pointer/CurrentActualValues[4]
//     Term 163 (AT2000-0250)/CC Inputs/Current actual value Ch.6 <-> Data Pointer/CurrentActualValues[5]
//     Term 163 (AT2000-0250)/CC Inputs/Current actual value Ch.7 <-> Data Pointer/CurrentActualValues[6]
//     Term 163 (AT2000-0250)/CC Inputs/Current actual value Ch.8 <-> Data Pointer/CurrentActualValues[7]
//     Term 163 (AT2000-0250)/CC Inputs/Current actual value Ch.9 <-> Data Pointer/CurrentActualValues[8]
//     Term 163 (AT2000-0250)/CC Inputs/Status <-> Data Pointer/Status
//     Term 163 (AT2000-0250)/CC Outputs/Control <-> Data Pointer/Control
//     Term 163 (AT2000-0250)/CC Outputs/Current setpoint value Ch.1 <-> Data Pointer/CurrentSetpointValues[0]
//     Term 163 (AT2000-0250)/CC Outputs/Current setpoint value Ch.10 <-> Data Pointer/CurrentSetpointValues[9]
//     Term 163 (AT2000-0250)/CC Outputs/Current setpoint value Ch.11 <-> Data Pointer/CurrentSetpointValues[10]
//     Term 163 (AT2000-0250)/CC Outputs/Current setpoint value Ch.12 <-> Data Pointer/CurrentSetpointValues[11]
//     Term 163 (AT2000-0250)/CC Outputs/Current setpoint value Ch.13 <-> Data Pointer/CurrentSetpointValues[12]
//     Term 163 (AT2000-0250)/CC Outputs/Current setpoint value Ch.14 <-> Data Pointer/CurrentSetpointValues[13]
//     Term 163 (AT2000-0250)/CC Outputs/Current setpoint value Ch.15 <-> Data Pointer/CurrentSetpointValues[14]
//     Term 163 (AT2000-0250)/CC Outputs/Current setpoint value Ch.2 <-> Data Pointer/CurrentSetpointValues[1]
//     Term 163 (AT2000-0250)/CC Outputs/Current setpoint value Ch.3 <-> Data Pointer/CurrentSetpointValues[2]
//     Term 163 (AT2000-0250)/CC Outputs/Current setpoint value Ch.4 <-> Data Pointer/CurrentSetpointValues[3]
//     Term 163 (AT2000-0250)/CC Outputs/Current setpoint value Ch.5 <-> Data Pointer/CurrentSetpointValues[4]
//     Term 163 (AT2000-0250)/CC Outputs/Current setpoint value Ch.6 <-> Data Pointer/CurrentSetpointValues[5]
//     Term 163 (AT2000-0250)/CC Outputs/Current setpoint value Ch.7 <-> Data Pointer/CurrentSetpointValues[6]
//     Term 163 (AT2000-0250)/CC Outputs/Current setpoint value Ch.8 <-> Data Pointer/CurrentSetpointValues[7]
//     Term 163 (AT2000-0250)/CC Outputs/Current setpoint value Ch.9 <-> Data Pointer/CurrentSetpointValues[8]
//     Term 163 (AT2000-0250)/Term 164 (AT2000-5250)/FB Inputs/Value Channel 01 <-> Data Pointer/RawPositionValues[0]
//     Term 163 (AT2000-0250)/Term 164 (AT2000-5250)/FB Inputs/Value Channel 02 <-> Data Pointer/RawPositionValues[1]
//     Term 163 (AT2000-0250)/Term 164 (AT2000-5250)/FB Inputs/Value Channel 03 <-> Data Pointer/RawPositionValues[2]
//     Term 163 (AT2000-0250)/Term 164 (AT2000-5250)/FB Inputs/Value Channel 04 <-> Data Pointer/RawPositionValues[3]
//     Term 163 (AT2000-0250)/Term 164 (AT2000-5250)/FB Inputs/Value Channel 05 <-> Data Pointer/RawPositionValues[4]
//     Term 163 (AT2000-0250)/Term 164 (AT2000-5250)/FB Inputs/Value Channel 06 <-> Data Pointer/RawPositionValues[5]
//     Term 163 (AT2000-0250)/Term 164 (AT2000-5250)/FB Inputs/Value Channel 07 <-> Data Pointer/RawPositionValues[6]
//     Term 163 (AT2000-0250)/Term 164 (AT2000-5250)/FB Inputs/Value Channel 08 <-> Data Pointer/RawPositionValues[7]
//     Term 163 (AT2000-0250)/Term 164 (AT2000-5250)/FB Inputs/Value Channel 09 <-> Data Pointer/RawPositionValues[8]
//     Term 163 (AT2000-0250)/Term 164 (AT2000-5250)/FB Inputs/Value Channel 10 <-> Data Pointer/RawPositionValues[9]
//     Term 163 (AT2000-0250)/Term 164 (AT2000-5250)/FB Inputs/Value Channel 11 <-> Data Pointer/RawPositionValues[10]
//     Term 163 (AT2000-0250)/Term 164 (AT2000-5250)/FB Inputs/Value Channel 12 <-> Data Pointer/RawPositionValues[11]
//     Term 163 (AT2000-0250)/Term 164 (AT2000-5250)/FB Inputs/Value Channel 13 <-> Data Pointer/RawPositionValues[12]
//     Term 163 (AT2000-0250)/Term 164 (AT2000-5250)/FB Inputs/Value Channel 14 <-> Data Pointer/RawPositionValues[13]
//     Term 163 (AT2000-0250)/Term 164 (AT2000-5250)/FB Inputs/Value Channel 15 <-> Data Pointer/RawPositionValues[14]
//     Term 163 (AT2000-0250)/Term 164 (AT2000-5250)/FB Inputs/Value Channel 16 <-> Data Pointer/RawPositionValues[15]
//     Term 163 (AT2000-0250)/Term 164 (AT2000-5250)/FB Inputs/Value Channel 17 <-> Data Pointer/RawPositionValues[16]
//     Term 163 (AT2000-0250)/Term 164 (AT2000-5250)/FB Inputs/Value Channel 18 <-> Data Pointer/RawPositionValues[17]
//     Term 163 (AT2000-0250)/Term 164 (AT2000-5250)/FB Inputs/Value Channel 19 <-> Data Pointer/RawPositionValues[18]
//     Term 163 (AT2000-0250)/Term 164 (AT2000-5250)/FB Inputs/Value Channel 20 <-> Data Pointer/RawPositionValues[19]
//     Term 163 (AT2000-0250)/Term 164 (AT2000-5250)/FB Inputs/Value Channel 21 <-> Data Pointer/RawPositionValues[20]
//     Term 163 (AT2000-0250)/Term 164 (AT2000-5250)/FB Inputs/Value Channel 22 <-> Data Pointer/RawPositionValues[21]
//     Term 163 (AT2000-0250)/Term 164 (AT2000-5250)/FB Inputs/Value Channel 23 <-> Data Pointer/RawPositionValues[22]
//     Term 163 (AT2000-0250)/Term 164 (AT2000-5250)/FB Inputs/Value Channel 24 <-> Data Pointer/RawPositionValues[23]
//     Term 163 (AT2000-0250)/Term 164 (AT2000-5250)/FB Inputs/Value Channel 25 <-> Data Pointer/RawPositionValues[24]
//     Term 163 (AT2000-0250)/Term 164 (AT2000-5250)/FB Inputs/Value Channel 26 <-> Data Pointer/RawPositionValues[25]
//     Term 163 (AT2000-0250)/Term 164 (AT2000-5250)/FB Inputs/Value Channel 27 <-> Data Pointer/RawPositionValues[26]
//     Term 163 (AT2000-0250)/Term 164 (AT2000-5250)/FB Inputs/Value Channel 28 <-> Data Pointer/RawPositionValues[27]
//     Term 163 (AT2000-0250)/Term 164 (AT2000-5250)/FB Inputs/Value Channel 29 <-> Data Pointer/RawPositionValues[28]
//     Term 163 (AT2000-0250)/Term 164 (AT2000-5250)/FB Inputs/Value Channel 30 <-> Data Pointer/RawPositionValues[29]
//     Term 163 (AT2000-0250)/Term 164 (AT2000-5250)/FB Inputs/Value Channel 31 <-> Data Pointer/RawPositionValues[30]
//     Term 163 (AT2000-0250)/Term 164 (AT2000-5250)/FB Inputs/Value Channel 32 <-> Data Pointer/RawPositionValues[31]
//   Device 2 <-> TcCOM Objects/XTS ProcessingUnit 1/Part 1/Module 5
//     Term 9 (AT2002-0250)/CC Inputs/Current actual value Ch.1 <-> Data Pointer/CurrentActualValues[0]
//     Term 9 (AT2002-0250)/CC Inputs/Current actual value Ch.10 <-> Data Pointer/CurrentActualValues[9]
//     Term 9 (AT2002-0250)/CC Inputs/Current actual value Ch.11 <-> Data Pointer/CurrentActualValues[10]
//     Term 9 (AT2002-0250)/CC Inputs/Current actual value Ch.12 <-> Data Pointer/CurrentActualValues[11]
//     Term 9 (AT2002-0250)/CC Inputs/Current actual value Ch.13 <-> Data Pointer/CurrentActualValues[12]
//     Term 9 (AT2002-0250)/CC Inputs/Current actual value Ch.14 <-> Data Pointer/CurrentActualValues[13]
//     Term 9 (AT2002-0250)/CC Inputs/Current actual value Ch.15 <-> Data Pointer/CurrentActualValues[14]
//     Term 9 (AT2002-0250)/CC Inputs/Current actual value Ch.2 <-> Data Pointer/CurrentActualValues[1]
//     Term 9 (AT2002-0250)/CC Inputs/Current actual value Ch.3 <-> Data Pointer/CurrentActualValues[2]
//     Term 9 (AT2002-0250)/CC Inputs/Current actual value Ch.4 <-> Data Pointer/CurrentActualValues[3]
//     Term 9 (AT2002-0250)/CC Inputs/Current actual value Ch.5 <-> Data Pointer/CurrentActualValues[4]
//     Term 9 (AT2002-0250)/CC Inputs/Current actual value Ch.6 <-> Data Pointer/CurrentActualValues[5]
//     Term 9 (AT2002-0250)/CC Inputs/Current actual value Ch.7 <-> Data Pointer/CurrentActualValues[6]
//     Term 9 (AT2002-0250)/CC Inputs/Current actual value Ch.8 <-> Data Pointer/CurrentActualValues[7]
//     Term 9 (AT2002-0250)/CC Inputs/Current actual value Ch.9 <-> Data Pointer/CurrentActualValues[8]
//     Term 9 (AT2002-0250)/CC Inputs/Status <-> Data Pointer/Status
//     Term 9 (AT2002-0250)/CC Outputs/Control <-> Data Pointer/Control
//     Term 9 (AT2002-0250)/CC Outputs/Current setpoint value Ch.1 <-> Data Pointer/CurrentSetpointValues[0]
//     Term 9 (AT2002-0250)/CC Outputs/Current setpoint value Ch.10 <-> Data Pointer/CurrentSetpointValues[9]
//     Term 9 (AT2002-0250)/CC Outputs/Current setpoint value Ch.11 <-> Data Pointer/CurrentSetpointValues[10]
//     Term 9 (AT2002-0250)/CC Outputs/Current setpoint value Ch.12 <-> Data Pointer/CurrentSetpointValues[11]
//     Term 9 (AT2002-0250)/CC Outputs/Current setpoint value Ch.13 <-> Data Pointer/CurrentSetpointValues[12]
//     Term 9 (AT2002-0250)/CC Outputs/Current setpoint value Ch.14 <-> Data Pointer/CurrentSetpointValues[13]
//     Term 9 (AT2002-0250)/CC Outputs/Current setpoint value Ch.15 <-> Data Pointer/CurrentSetpointValues[14]
//     Term 9 (AT2002-0250)/CC Outputs/Current setpoint value Ch.2 <-> Data Pointer/CurrentSetpointValues[1]
//     Term 9 (AT2002-0250)/CC Outputs/Current setpoint value Ch.3 <-> Data Pointer/CurrentSetpointValues[2]
//     Term 9 (AT2002-0250)/CC Outputs/Current setpoint value Ch.4 <-> Data Pointer/CurrentSetpointValues[3]
//     Term 9 (AT2002-0250)/CC Outputs/Current setpoint value Ch.5 <-> Data Pointer/CurrentSetpointValues[4]
//     Term 9 (AT2002-0250)/CC Outputs/Current setpoint value Ch.6 <-> Data Pointer/CurrentSetpointValues[5]
//     Term 9 (AT2002-0250)/CC Outputs/Current setpoint value Ch.7 <-> Data Pointer/CurrentSetpointValues[6]
//     Term 9 (AT2002-0250)/CC Outputs/Current setpoint value Ch.8 <-> Data Pointer/CurrentSetpointValues[7]
//     Term 9 (AT2002-0250)/CC Outputs/Current setpoint value Ch.9 <-> Data Pointer/CurrentSetpointValues[8]
//     Term 9 (AT2002-0250)/Term 10 (AT2002-5250)/FB Inputs/Value Channel 01 <-> Data Pointer/RawPositionValues[0]
//     Term 9 (AT2002-0250)/Term 10 (AT2002-5250)/FB Inputs/Value Channel 02 <-> Data Pointer/RawPositionValues[1]
//     Term 9 (AT2002-0250)/Term 10 (AT2002-5250)/FB Inputs/Value Channel 03 <-> Data Pointer/RawPositionValues[2]
//     Term 9 (AT2002-0250)/Term 10 (AT2002-5250)/FB Inputs/Value Channel 04 <-> Data Pointer/RawPositionValues[3]
//     Term 9 (AT2002-0250)/Term 10 (AT2002-5250)/FB Inputs/Value Channel 05 <-> Data Pointer/RawPositionValues[4]
//     Term 9 (AT2002-0250)/Term 10 (AT2002-5250)/FB Inputs/Value Channel 06 <-> Data Pointer/RawPositionValues[5]
//     Term 9 (AT2002-0250)/Term 10 (AT2002-5250)/FB Inputs/Value Channel 07 <-> Data Pointer/RawPositionValues[6]
//     Term 9 (AT2002-0250)/Term 10 (AT2002-5250)/FB Inputs/Value Channel 08 <-> Data Pointer/RawPositionValues[7]
//     Term 9 (AT2002-0250)/Term 10 (AT2002-5250)/FB Inputs/Value Channel 09 <-> Data Pointer/RawPositionValues[8]
//     Term 9 (AT2002-0250)/Term 10 (AT2002-5250)/FB Inputs/Value Channel 10 <-> Data Pointer/RawPositionValues[9]
//     Term 9 (AT2002-0250)/Term 10 (AT2002-5250)/FB Inputs/Value Channel 11 <-> Data Pointer/RawPositionValues[10]
//     Term 9 (AT2002-0250)/Term 10 (AT2002-5250)/FB Inputs/Value Channel 12 <-> Data Pointer/RawPositionValues[11]
//     Term 9 (AT2002-0250)/Term 10 (AT2002-5250)/FB Inputs/Value Channel 13 <-> Data Pointer/RawPositionValues[12]
//     Term 9 (AT2002-0250)/Term 10 (AT2002-5250)/FB Inputs/Value Channel 14 <-> Data Pointer/RawPositionValues[13]
//     Term 9 (AT2002-0250)/Term 10 (AT2002-5250)/FB Inputs/Value Channel 15 <-> Data Pointer/RawPositionValues[14]
//     Term 9 (AT2002-0250)/Term 10 (AT2002-5250)/FB Inputs/Value Channel 16 <-> Data Pointer/RawPositionValues[15]
//     Term 9 (AT2002-0250)/Term 10 (AT2002-5250)/FB Inputs/Value Channel 17 <-> Data Pointer/RawPositionValues[16]
//     Term 9 (AT2002-0250)/Term 10 (AT2002-5250)/FB Inputs/Value Channel 18 <-> Data Pointer/RawPositionValues[17]
//     Term 9 (AT2002-0250)/Term 10 (AT2002-5250)/FB Inputs/Value Channel 19 <-> Data Pointer/RawPositionValues[18]
//     Term 9 (AT2002-0250)/Term 10 (AT2002-5250)/FB Inputs/Value Channel 20 <-> Data Pointer/RawPositionValues[19]
//     Term 9 (AT2002-0250)/Term 10 (AT2002-5250)/FB Inputs/Value Channel 21 <-> Data Pointer/RawPositionValues[20]
//     Term 9 (AT2002-0250)/Term 10 (AT2002-5250)/FB Inputs/Value Channel 22 <-> Data Pointer/RawPositionValues[21]
//     Term 9 (AT2002-0250)/Term 10 (AT2002-5250)/FB Inputs/Value Channel 23 <-> Data Pointer/RawPositionValues[22]
//     Term 9 (AT2002-0250)/Term 10 (AT2002-5250)/FB Inputs/Value Channel 24 <-> Data Pointer/RawPositionValues[23]
//     Term 9 (AT2002-0250)/Term 10 (AT2002-5250)/FB Inputs/Value Channel 25 <-> Data Pointer/RawPositionValues[24]
//     Term 9 (AT2002-0250)/Term 10 (AT2002-5250)/FB Inputs/Value Channel 26 <-> Data Pointer/RawPositionValues[25]
//     Term 9 (AT2002-0250)/Term 10 (AT2002-5250)/FB Inputs/Value Channel 27 <-> Data Pointer/RawPositionValues[26]
//     Term 9 (AT2002-0250)/Term 10 (AT2002-5250)/FB Inputs/Value Channel 28 <-> Data Pointer/RawPositionValues[27]
//     Term 9 (AT2002-0250)/Term 10 (AT2002-5250)/FB Inputs/Value Channel 29 <-> Data Pointer/RawPositionValues[28]
//     Term 9 (AT2002-0250)/Term 10 (AT2002-5250)/FB Inputs/Value Channel 30 <-> Data Pointer/RawPositionValues[29]
//     Term 9 (AT2002-0250)/Term 10 (AT2002-5250)/FB Inputs/Value Channel 31 <-> Data Pointer/RawPositionValues[30]
//     Term 9 (AT2002-0250)/Term 10 (AT2002-5250)/FB Inputs/Value Channel 32 <-> Data Pointer/RawPositionValues[31]
//   Device 2 <-> TcCOM Objects/XTS ProcessingUnit 1/Part 1/Module 6
//     Term 11 (AT2000-0250)/CC Inputs/Current actual value Ch.1 <-> Data Pointer/CurrentActualValues[0]
//     Term 11 (AT2000-0250)/CC Inputs/Current actual value Ch.10 <-> Data Pointer/CurrentActualValues[9]
//     Term 11 (AT2000-0250)/CC Inputs/Current actual value Ch.11 <-> Data Pointer/CurrentActualValues[10]
//     Term 11 (AT2000-0250)/CC Inputs/Current actual value Ch.12 <-> Data Pointer/CurrentActualValues[11]
//     Term 11 (AT2000-0250)/CC Inputs/Current actual value Ch.13 <-> Data Pointer/CurrentActualValues[12]
//     Term 11 (AT2000-0250)/CC Inputs/Current actual value Ch.14 <-> Data Pointer/CurrentActualValues[13]
//     Term 11 (AT2000-0250)/CC Inputs/Current actual value Ch.15 <-> Data Pointer/CurrentActualValues[14]
//     Term 11 (AT2000-0250)/CC Inputs/Current actual value Ch.2 <-> Data Pointer/CurrentActualValues[1]
//     Term 11 (AT2000-0250)/CC Inputs/Current actual value Ch.3 <-> Data Pointer/CurrentActualValues[2]
//     Term 11 (AT2000-0250)/CC Inputs/Current actual value Ch.4 <-> Data Pointer/CurrentActualValues[3]
//     Term 11 (AT2000-0250)/CC Inputs/Current actual value Ch.5 <-> Data Pointer/CurrentActualValues[4]
//     Term 11 (AT2000-0250)/CC Inputs/Current actual value Ch.6 <-> Data Pointer/CurrentActualValues[5]
//     Term 11 (AT2000-0250)/CC Inputs/Current actual value Ch.7 <-> Data Pointer/CurrentActualValues[6]
//     Term 11 (AT2000-0250)/CC Inputs/Current actual value Ch.8 <-> Data Pointer/CurrentActualValues[7]
//     Term 11 (AT2000-0250)/CC Inputs/Current actual value Ch.9 <-> Data Pointer/CurrentActualValues[8]
//     Term 11 (AT2000-0250)/CC Inputs/Status <-> Data Pointer/Status
//     Term 11 (AT2000-0250)/CC Outputs/Control <-> Data Pointer/Control
//     Term 11 (AT2000-0250)/CC Outputs/Current setpoint value Ch.1 <-> Data Pointer/CurrentSetpointValues[0]
//     Term 11 (AT2000-0250)/CC Outputs/Current setpoint value Ch.10 <-> Data Pointer/CurrentSetpointValues[9]
//     Term 11 (AT2000-0250)/CC Outputs/Current setpoint value Ch.11 <-> Data Pointer/CurrentSetpointValues[10]
//     Term 11 (AT2000-0250)/CC Outputs/Current setpoint value Ch.12 <-> Data Pointer/CurrentSetpointValues[11]
//     Term 11 (AT2000-0250)/CC Outputs/Current setpoint value Ch.13 <-> Data Pointer/CurrentSetpointValues[12]
//     Term 11 (AT2000-0250)/CC Outputs/Current setpoint value Ch.14 <-> Data Pointer/CurrentSetpointValues[13]
//     Term 11 (AT2000-0250)/CC Outputs/Current setpoint value Ch.15 <-> Data Pointer/CurrentSetpointValues[14]
//     Term 11 (AT2000-0250)/CC Outputs/Current setpoint value Ch.2 <-> Data Pointer/CurrentSetpointValues[1]
//     Term 11 (AT2000-0250)/CC Outputs/Current setpoint value Ch.3 <-> Data Pointer/CurrentSetpointValues[2]
//     Term 11 (AT2000-0250)/CC Outputs/Current setpoint value Ch.4 <-> Data Pointer/CurrentSetpointValues[3]
//     Term 11 (AT2000-0250)/CC Outputs/Current setpoint value Ch.5 <-> Data Pointer/CurrentSetpointValues[4]
//     Term 11 (AT2000-0250)/CC Outputs/Current setpoint value Ch.6 <-> Data Pointer/CurrentSetpointValues[5]
//     Term 11 (AT2000-0250)/CC Outputs/Current setpoint value Ch.7 <-> Data Pointer/CurrentSetpointValues[6]
//     Term 11 (AT2000-0250)/CC Outputs/Current setpoint value Ch.8 <-> Data Pointer/CurrentSetpointValues[7]
//     Term 11 (AT2000-0250)/CC Outputs/Current setpoint value Ch.9 <-> Data Pointer/CurrentSetpointValues[8]
//     Term 11 (AT2000-0250)/Term 12 (AT2000-5250)/FB Inputs/Value Channel 01 <-> Data Pointer/RawPositionValues[0]
//     Term 11 (AT2000-0250)/Term 12 (AT2000-5250)/FB Inputs/Value Channel 02 <-> Data Pointer/RawPositionValues[1]
//     Term 11 (AT2000-0250)/Term 12 (AT2000-5250)/FB Inputs/Value Channel 03 <-> Data Pointer/RawPositionValues[2]
//     Term 11 (AT2000-0250)/Term 12 (AT2000-5250)/FB Inputs/Value Channel 04 <-> Data Pointer/RawPositionValues[3]
//     Term 11 (AT2000-0250)/Term 12 (AT2000-5250)/FB Inputs/Value Channel 05 <-> Data Pointer/RawPositionValues[4]
//     Term 11 (AT2000-0250)/Term 12 (AT2000-5250)/FB Inputs/Value Channel 06 <-> Data Pointer/RawPositionValues[5]
//     Term 11 (AT2000-0250)/Term 12 (AT2000-5250)/FB Inputs/Value Channel 07 <-> Data Pointer/RawPositionValues[6]
//     Term 11 (AT2000-0250)/Term 12 (AT2000-5250)/FB Inputs/Value Channel 08 <-> Data Pointer/RawPositionValues[7]
//     Term 11 (AT2000-0250)/Term 12 (AT2000-5250)/FB Inputs/Value Channel 09 <-> Data Pointer/RawPositionValues[8]
//     Term 11 (AT2000-0250)/Term 12 (AT2000-5250)/FB Inputs/Value Channel 10 <-> Data Pointer/RawPositionValues[9]
//     Term 11 (AT2000-0250)/Term 12 (AT2000-5250)/FB Inputs/Value Channel 11 <-> Data Pointer/RawPositionValues[10]
//     Term 11 (AT2000-0250)/Term 12 (AT2000-5250)/FB Inputs/Value Channel 12 <-> Data Pointer/RawPositionValues[11]
//     Term 11 (AT2000-0250)/Term 12 (AT2000-5250)/FB Inputs/Value Channel 13 <-> Data Pointer/RawPositionValues[12]
//     Term 11 (AT2000-0250)/Term 12 (AT2000-5250)/FB Inputs/Value Channel 14 <-> Data Pointer/RawPositionValues[13]
//     Term 11 (AT2000-0250)/Term 12 (AT2000-5250)/FB Inputs/Value Channel 15 <-> Data Pointer/RawPositionValues[14]
//     Term 11 (AT2000-0250)/Term 12 (AT2000-5250)/FB Inputs/Value Channel 16 <-> Data Pointer/RawPositionValues[15]
//     Term 11 (AT2000-0250)/Term 12 (AT2000-5250)/FB Inputs/Value Channel 17 <-> Data Pointer/RawPositionValues[16]
//     Term 11 (AT2000-0250)/Term 12 (AT2000-5250)/FB Inputs/Value Channel 18 <-> Data Pointer/RawPositionValues[17]
//     Term 11 (AT2000-0250)/Term 12 (AT2000-5250)/FB Inputs/Value Channel 19 <-> Data Pointer/RawPositionValues[18]
//     Term 11 (AT2000-0250)/Term 12 (AT2000-5250)/FB Inputs/Value Channel 20 <-> Data Pointer/RawPositionValues[19]
//     Term 11 (AT2000-0250)/Term 12 (AT2000-5250)/FB Inputs/Value Channel 21 <-> Data Pointer/RawPositionValues[20]
//     Term 11 (AT2000-0250)/Term 12 (AT2000-5250)/FB Inputs/Value Channel 22 <-> Data Pointer/RawPositionValues[21]
//     Term 11 (AT2000-0250)/Term 12 (AT2000-5250)/FB Inputs/Value Channel 23 <-> Data Pointer/RawPositionValues[22]
//     Term 11 (AT2000-0250)/Term 12 (AT2000-5250)/FB Inputs/Value Channel 24 <-> Data Pointer/RawPositionValues[23]
//     Term 11 (AT2000-0250)/Term 12 (AT2000-5250)/FB Inputs/Value Channel 25 <-> Data Pointer/RawPositionValues[24]
//     Term 11 (AT2000-0250)/Term 12 (AT2000-5250)/FB Inputs/Value Channel 26 <-> Data Pointer/RawPositionValues[25]
//     Term 11 (AT2000-0250)/Term 12 (AT2000-5250)/FB Inputs/Value Channel 27 <-> Data Pointer/RawPositionValues[26]
//     Term 11 (AT2000-0250)/Term 12 (AT2000-5250)/FB Inputs/Value Channel 28 <-> Data Pointer/RawPositionValues[27]
//     Term 11 (AT2000-0250)/Term 12 (AT2000-5250)/FB Inputs/Value Channel 29 <-> Data Pointer/RawPositionValues[28]
//     Term 11 (AT2000-0250)/Term 12 (AT2000-5250)/FB Inputs/Value Channel 30 <-> Data Pointer/RawPositionValues[29]
//     Term 11 (AT2000-0250)/Term 12 (AT2000-5250)/FB Inputs/Value Channel 31 <-> Data Pointer/RawPositionValues[30]
//     Term 11 (AT2000-0250)/Term 12 (AT2000-5250)/FB Inputs/Value Channel 32 <-> Data Pointer/RawPositionValues[31]
//   Device 2 <-> TcCOM Objects/XTS ProcessingUnit 1/Part 1/Module 7
//     Term 13 (AT2000-0250)/CC Inputs/Current actual value Ch.1 <-> Data Pointer/CurrentActualValues[0]
//     Term 13 (AT2000-0250)/CC Inputs/Current actual value Ch.10 <-> Data Pointer/CurrentActualValues[9]
//     Term 13 (AT2000-0250)/CC Inputs/Current actual value Ch.11 <-> Data Pointer/CurrentActualValues[10]
//     Term 13 (AT2000-0250)/CC Inputs/Current actual value Ch.12 <-> Data Pointer/CurrentActualValues[11]
//     Term 13 (AT2000-0250)/CC Inputs/Current actual value Ch.13 <-> Data Pointer/CurrentActualValues[12]
//     Term 13 (AT2000-0250)/CC Inputs/Current actual value Ch.14 <-> Data Pointer/CurrentActualValues[13]
//     Term 13 (AT2000-0250)/CC Inputs/Current actual value Ch.15 <-> Data Pointer/CurrentActualValues[14]
//     Term 13 (AT2000-0250)/CC Inputs/Current actual value Ch.2 <-> Data Pointer/CurrentActualValues[1]
//     Term 13 (AT2000-0250)/CC Inputs/Current actual value Ch.3 <-> Data Pointer/CurrentActualValues[2]
//     Term 13 (AT2000-0250)/CC Inputs/Current actual value Ch.4 <-> Data Pointer/CurrentActualValues[3]
//     Term 13 (AT2000-0250)/CC Inputs/Current actual value Ch.5 <-> Data Pointer/CurrentActualValues[4]
//     Term 13 (AT2000-0250)/CC Inputs/Current actual value Ch.6 <-> Data Pointer/CurrentActualValues[5]
//     Term 13 (AT2000-0250)/CC Inputs/Current actual value Ch.7 <-> Data Pointer/CurrentActualValues[6]
//     Term 13 (AT2000-0250)/CC Inputs/Current actual value Ch.8 <-> Data Pointer/CurrentActualValues[7]
//     Term 13 (AT2000-0250)/CC Inputs/Current actual value Ch.9 <-> Data Pointer/CurrentActualValues[8]
//     Term 13 (AT2000-0250)/CC Inputs/Status <-> Data Pointer/Status
//     Term 13 (AT2000-0250)/CC Outputs/Control <-> Data Pointer/Control
//     Term 13 (AT2000-0250)/CC Outputs/Current setpoint value Ch.1 <-> Data Pointer/CurrentSetpointValues[0]
//     Term 13 (AT2000-0250)/CC Outputs/Current setpoint value Ch.10 <-> Data Pointer/CurrentSetpointValues[9]
//     Term 13 (AT2000-0250)/CC Outputs/Current setpoint value Ch.11 <-> Data Pointer/CurrentSetpointValues[10]
//     Term 13 (AT2000-0250)/CC Outputs/Current setpoint value Ch.12 <-> Data Pointer/CurrentSetpointValues[11]
//     Term 13 (AT2000-0250)/CC Outputs/Current setpoint value Ch.13 <-> Data Pointer/CurrentSetpointValues[12]
//     Term 13 (AT2000-0250)/CC Outputs/Current setpoint value Ch.14 <-> Data Pointer/CurrentSetpointValues[13]
//     Term 13 (AT2000-0250)/CC Outputs/Current setpoint value Ch.15 <-> Data Pointer/CurrentSetpointValues[14]
//     Term 13 (AT2000-0250)/CC Outputs/Current setpoint value Ch.2 <-> Data Pointer/CurrentSetpointValues[1]
//     Term 13 (AT2000-0250)/CC Outputs/Current setpoint value Ch.3 <-> Data Pointer/CurrentSetpointValues[2]
//     Term 13 (AT2000-0250)/CC Outputs/Current setpoint value Ch.4 <-> Data Pointer/CurrentSetpointValues[3]
//     Term 13 (AT2000-0250)/CC Outputs/Current setpoint value Ch.5 <-> Data Pointer/CurrentSetpointValues[4]
//     Term 13 (AT2000-0250)/CC Outputs/Current setpoint value Ch.6 <-> Data Pointer/CurrentSetpointValues[5]
//     Term 13 (AT2000-0250)/CC Outputs/Current setpoint value Ch.7 <-> Data Pointer/CurrentSetpointValues[6]
//     Term 13 (AT2000-0250)/CC Outputs/Current setpoint value Ch.8 <-> Data Pointer/CurrentSetpointValues[7]
//     Term 13 (AT2000-0250)/CC Outputs/Current setpoint value Ch.9 <-> Data Pointer/CurrentSetpointValues[8]
//     Term 13 (AT2000-0250)/Term 14 (AT2000-5250)/FB Inputs/Value Channel 01 <-> Data Pointer/RawPositionValues[0]
//     Term 13 (AT2000-0250)/Term 14 (AT2000-5250)/FB Inputs/Value Channel 02 <-> Data Pointer/RawPositionValues[1]
//     Term 13 (AT2000-0250)/Term 14 (AT2000-5250)/FB Inputs/Value Channel 03 <-> Data Pointer/RawPositionValues[2]
//     Term 13 (AT2000-0250)/Term 14 (AT2000-5250)/FB Inputs/Value Channel 04 <-> Data Pointer/RawPositionValues[3]
//     Term 13 (AT2000-0250)/Term 14 (AT2000-5250)/FB Inputs/Value Channel 05 <-> Data Pointer/RawPositionValues[4]
//     Term 13 (AT2000-0250)/Term 14 (AT2000-5250)/FB Inputs/Value Channel 06 <-> Data Pointer/RawPositionValues[5]
//     Term 13 (AT2000-0250)/Term 14 (AT2000-5250)/FB Inputs/Value Channel 07 <-> Data Pointer/RawPositionValues[6]
//     Term 13 (AT2000-0250)/Term 14 (AT2000-5250)/FB Inputs/Value Channel 08 <-> Data Pointer/RawPositionValues[7]
//     Term 13 (AT2000-0250)/Term 14 (AT2000-5250)/FB Inputs/Value Channel 09 <-> Data Pointer/RawPositionValues[8]
//     Term 13 (AT2000-0250)/Term 14 (AT2000-5250)/FB Inputs/Value Channel 10 <-> Data Pointer/RawPositionValues[9]
//     Term 13 (AT2000-0250)/Term 14 (AT2000-5250)/FB Inputs/Value Channel 11 <-> Data Pointer/RawPositionValues[10]
//     Term 13 (AT2000-0250)/Term 14 (AT2000-5250)/FB Inputs/Value Channel 12 <-> Data Pointer/RawPositionValues[11]
//     Term 13 (AT2000-0250)/Term 14 (AT2000-5250)/FB Inputs/Value Channel 13 <-> Data Pointer/RawPositionValues[12]
//     Term 13 (AT2000-0250)/Term 14 (AT2000-5250)/FB Inputs/Value Channel 14 <-> Data Pointer/RawPositionValues[13]
//     Term 13 (AT2000-0250)/Term 14 (AT2000-5250)/FB Inputs/Value Channel 15 <-> Data Pointer/RawPositionValues[14]
//     Term 13 (AT2000-0250)/Term 14 (AT2000-5250)/FB Inputs/Value Channel 16 <-> Data Pointer/RawPositionValues[15]
//     Term 13 (AT2000-0250)/Term 14 (AT2000-5250)/FB Inputs/Value Channel 17 <-> Data Pointer/RawPositionValues[16]
//     Term 13 (AT2000-0250)/Term 14 (AT2000-5250)/FB Inputs/Value Channel 18 <-> Data Pointer/RawPositionValues[17]
//     Term 13 (AT2000-0250)/Term 14 (AT2000-5250)/FB Inputs/Value Channel 19 <-> Data Pointer/RawPositionValues[18]
//     Term 13 (AT2000-0250)/Term 14 (AT2000-5250)/FB Inputs/Value Channel 20 <-> Data Pointer/RawPositionValues[19]
//     Term 13 (AT2000-0250)/Term 14 (AT2000-5250)/FB Inputs/Value Channel 21 <-> Data Pointer/RawPositionValues[20]
//     Term 13 (AT2000-0250)/Term 14 (AT2000-5250)/FB Inputs/Value Channel 22 <-> Data Pointer/RawPositionValues[21]
//     Term 13 (AT2000-0250)/Term 14 (AT2000-5250)/FB Inputs/Value Channel 23 <-> Data Pointer/RawPositionValues[22]
//     Term 13 (AT2000-0250)/Term 14 (AT2000-5250)/FB Inputs/Value Channel 24 <-> Data Pointer/RawPositionValues[23]
//     Term 13 (AT2000-0250)/Term 14 (AT2000-5250)/FB Inputs/Value Channel 25 <-> Data Pointer/RawPositionValues[24]
//     Term 13 (AT2000-0250)/Term 14 (AT2000-5250)/FB Inputs/Value Channel 26 <-> Data Pointer/RawPositionValues[25]
//     Term 13 (AT2000-0250)/Term 14 (AT2000-5250)/FB Inputs/Value Channel 27 <-> Data Pointer/RawPositionValues[26]
//     Term 13 (AT2000-0250)/Term 14 (AT2000-5250)/FB Inputs/Value Channel 28 <-> Data Pointer/RawPositionValues[27]
//     Term 13 (AT2000-0250)/Term 14 (AT2000-5250)/FB Inputs/Value Channel 29 <-> Data Pointer/RawPositionValues[28]
//     Term 13 (AT2000-0250)/Term 14 (AT2000-5250)/FB Inputs/Value Channel 30 <-> Data Pointer/RawPositionValues[29]
//     Term 13 (AT2000-0250)/Term 14 (AT2000-5250)/FB Inputs/Value Channel 31 <-> Data Pointer/RawPositionValues[30]
//     Term 13 (AT2000-0250)/Term 14 (AT2000-5250)/FB Inputs/Value Channel 32 <-> Data Pointer/RawPositionValues[31]
//   Device 2 <-> TcCOM Objects/XTS ProcessingUnit 1/Part 1/Module 8
//     Term 15 (AT2000-0250)/CC Inputs/Current actual value Ch.1 <-> Data Pointer/CurrentActualValues[0]
//     Term 15 (AT2000-0250)/CC Inputs/Current actual value Ch.10 <-> Data Pointer/CurrentActualValues[9]
//     Term 15 (AT2000-0250)/CC Inputs/Current actual value Ch.11 <-> Data Pointer/CurrentActualValues[10]
//     Term 15 (AT2000-0250)/CC Inputs/Current actual value Ch.12 <-> Data Pointer/CurrentActualValues[11]
//     Term 15 (AT2000-0250)/CC Inputs/Current actual value Ch.13 <-> Data Pointer/CurrentActualValues[12]
//     Term 15 (AT2000-0250)/CC Inputs/Current actual value Ch.14 <-> Data Pointer/CurrentActualValues[13]
//     Term 15 (AT2000-0250)/CC Inputs/Current actual value Ch.15 <-> Data Pointer/CurrentActualValues[14]
//     Term 15 (AT2000-0250)/CC Inputs/Current actual value Ch.2 <-> Data Pointer/CurrentActualValues[1]
//     Term 15 (AT2000-0250)/CC Inputs/Current actual value Ch.3 <-> Data Pointer/CurrentActualValues[2]
//     Term 15 (AT2000-0250)/CC Inputs/Current actual value Ch.4 <-> Data Pointer/CurrentActualValues[3]
//     Term 15 (AT2000-0250)/CC Inputs/Current actual value Ch.5 <-> Data Pointer/CurrentActualValues[4]
//     Term 15 (AT2000-0250)/CC Inputs/Current actual value Ch.6 <-> Data Pointer/CurrentActualValues[5]
//     Term 15 (AT2000-0250)/CC Inputs/Current actual value Ch.7 <-> Data Pointer/CurrentActualValues[6]
//     Term 15 (AT2000-0250)/CC Inputs/Current actual value Ch.8 <-> Data Pointer/CurrentActualValues[7]
//     Term 15 (AT2000-0250)/CC Inputs/Current actual value Ch.9 <-> Data Pointer/CurrentActualValues[8]
//     Term 15 (AT2000-0250)/CC Inputs/Status <-> Data Pointer/Status
//     Term 15 (AT2000-0250)/CC Outputs/Control <-> Data Pointer/Control
//     Term 15 (AT2000-0250)/CC Outputs/Current setpoint value Ch.1 <-> Data Pointer/CurrentSetpointValues[0]
//     Term 15 (AT2000-0250)/CC Outputs/Current setpoint value Ch.10 <-> Data Pointer/CurrentSetpointValues[9]
//     Term 15 (AT2000-0250)/CC Outputs/Current setpoint value Ch.11 <-> Data Pointer/CurrentSetpointValues[10]
//     Term 15 (AT2000-0250)/CC Outputs/Current setpoint value Ch.12 <-> Data Pointer/CurrentSetpointValues[11]
//     Term 15 (AT2000-0250)/CC Outputs/Current setpoint value Ch.13 <-> Data Pointer/CurrentSetpointValues[12]
